Fanuc TP program (LS listing): CODE1_1.ls

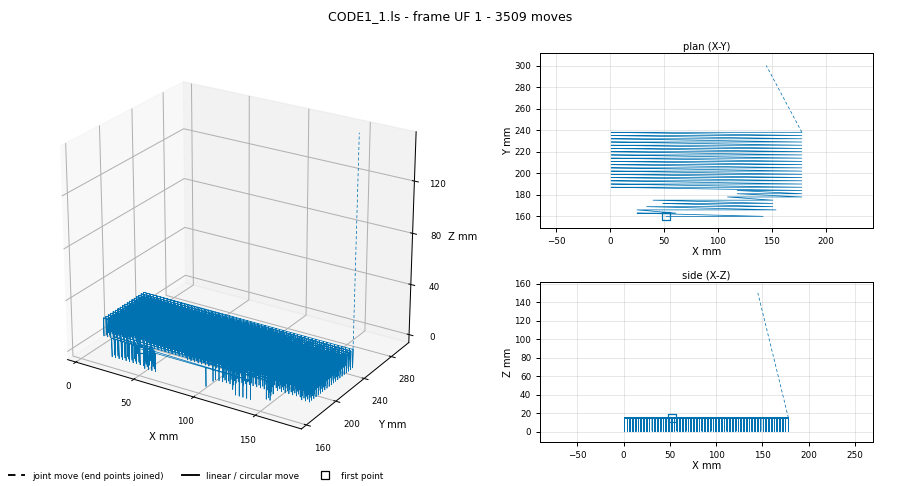
[picture p0: tool path of CODE1_1.ls in frame UF 1, 3509 of 3509 moves have a stored position in this frame; points joined in program order, loops and branches not executed]
/PROG CODE1_1
/ATTR
OWNER		= NOC_FANU;
COMMENT		= "NOC_FANUC";
PROG_SIZE	= 328;
CREATE		= DATE 97-07-08  TIME 03:05:20;
MODIFIED	= DATE 17-07-08  TIME 03:05:26;
FILE_NAME	= ;
VERSION		= 0;
LINE_COUNT	= 10;
MEMORY_SIZE	= 692;
PROTECT		= READ_WRITE;
TCD:  STACK_SIZE	= 0,
      TASK_PRIORITY	= 0,
      TIME_SLICE	= 0,
      BUSY_LAMP_OFF	= 0,
      ABORT_REQUEST	= 0,
      PAUSE_REQUEST	= 0;
DEFAULT_GROUP	= 1,*,*,*,*;
CONTROL_CODE	= 00000000 00000000;
/APPL
/MN
1:UFRAME_NUM=1 ;
2:UTOOL_NUM=1;
3:J P[7599] 10% CNT100;
4:L P[7600] 250mm/sec CNT100;
5:L P[7601] 250mm/sec FINE;
6:L P[7602] 250mm/sec CNT100;
7:L P[7603] 250mm/sec CNT100;
8:L P[7604] 250mm/sec FINE;
9:L P[7605] 250mm/sec CNT100;
10:L P[7606] 250mm/sec CNT100;
11:L P[7607] 250mm/sec FINE;
12:L P[7608] 250mm/sec CNT100;
13:L P[7609] 250mm/sec CNT100;
14:L P[7610] 250mm/sec FINE;
15:L P[7611] 250mm/sec CNT100;
16:L P[7612] 250mm/sec CNT100;
17:L P[7613] 250mm/sec FINE;
18:L P[7614] 250mm/sec CNT100;
19:L P[7636] 250mm/sec CNT100;
20:L P[7637] 250mm/sec FINE;
21:L P[7638] 250mm/sec CNT100;
22:L P[7639] 250mm/sec CNT100;
23:L P[7640] 250mm/sec FINE;
24:L P[7641] 250mm/sec CNT100;
25:L P[7642] 250mm/sec CNT100;
26:L P[7643] 250mm/sec FINE;
27:L P[7644] 250mm/sec CNT100;
28:L P[7645] 250mm/sec CNT100;
29:L P[7646] 250mm/sec FINE;
30:L P[7647] 250mm/sec CNT100;
31:L P[7648] 250mm/sec CNT100;
32:L P[7649] 250mm/sec FINE;
33:L P[7650] 250mm/sec CNT100;
34:L P[7666] 250mm/sec CNT100;
35:L P[7667] 250mm/sec FINE;
36:L P[7668] 250mm/sec CNT100;
37:L P[7669] 250mm/sec CNT100;
38:L P[7670] 250mm/sec FINE;
39:L P[7671] 250mm/sec CNT100;
40:L P[7672] 250mm/sec CNT100;
41:L P[7673] 250mm/sec FINE;
42:L P[7674] 250mm/sec CNT100;
43:L P[7675] 250mm/sec CNT100;
44:L P[7676] 250mm/sec FINE;
45:L P[7677] 250mm/sec CNT100;
46:L P[7678] 250mm/sec CNT100;
47:L P[7679] 250mm/sec FINE;
48:L P[7680] 250mm/sec CNT100;
49:L P[7681] 250mm/sec CNT100;
50:L P[7682] 250mm/sec FINE;
51:L P[7683] 250mm/sec CNT100;
52:L P[7684] 250mm/sec CNT100;
53:L P[7685] 250mm/sec FINE;
54:L P[7686] 250mm/sec CNT100;
55:L P[7687] 250mm/sec CNT100;
56:L P[7688] 250mm/sec FINE;
57:L P[7689] 250mm/sec CNT100;
58:L P[7690] 250mm/sec CNT100;
59:L P[7691] 250mm/sec FINE;
60:L P[7692] 250mm/sec CNT100;
61:L P[7693] 250mm/sec CNT100;
62:L P[7694] 250mm/sec FINE;
63:L P[7695] 250mm/sec CNT100;
64:L P[7696] 250mm/sec CNT100;
65:L P[7697] 250mm/sec FINE;
66:L P[7698] 250mm/sec CNT100;
67:L P[7702] 250mm/sec CNT100;
68:L P[7703] 250mm/sec FINE;
69:L P[7704] 250mm/sec CNT100;
70:L P[7756] 250mm/sec CNT100;
71:L P[7757] 250mm/sec FINE;
72:L P[7758] 250mm/sec CNT100;
73:L P[7759] 250mm/sec CNT100;
74:L P[7760] 250mm/sec FINE;
75:L P[7761] 250mm/sec CNT100;
76:L P[7762] 250mm/sec CNT100;
77:L P[7763] 250mm/sec FINE;
78:L P[7764] 250mm/sec CNT100;
79:L P[7765] 250mm/sec CNT100;
80:L P[7766] 250mm/sec FINE;
81:L P[7767] 250mm/sec CNT100;
82:L P[7768] 250mm/sec CNT100;
83:L P[7769] 250mm/sec FINE;
84:L P[7770] 250mm/sec CNT100;
85:L P[7771] 250mm/sec CNT100;
86:L P[7772] 250mm/sec FINE;
87:L P[7773] 250mm/sec CNT100;
88:L P[7774] 250mm/sec CNT100;
89:L P[7775] 250mm/sec FINE;
90:L P[7776] 250mm/sec CNT100;
91:L P[7777] 250mm/sec CNT100;
92:L P[7778] 250mm/sec FINE;
93:L P[7779] 250mm/sec CNT100;
94:L P[7783] 250mm/sec CNT100;
95:L P[7784] 250mm/sec FINE;
96:L P[7785] 250mm/sec CNT100;
97:L P[7786] 250mm/sec CNT100;
98:L P[7787] 250mm/sec FINE;
99:L P[7788] 250mm/sec CNT100;
100:L P[7789] 250mm/sec CNT100;
101:L P[7790] 250mm/sec FINE;
102:L P[7791] 250mm/sec CNT100;
103:L P[7810] 250mm/sec CNT100;
104:L P[7811] 250mm/sec FINE;
105:L P[7812] 250mm/sec CNT100;
106:L P[7837] 250mm/sec CNT100;
107:L P[7838] 250mm/sec FINE;
108:L P[7839] 250mm/sec CNT100;
109:L P[7840] 250mm/sec CNT100;
110:L P[7841] 250mm/sec FINE;
111:L P[7842] 250mm/sec CNT100;
112:L P[7849] 250mm/sec CNT100;
113:L P[7850] 250mm/sec FINE;
114:L P[7851] 250mm/sec CNT100;
115:L P[7855] 250mm/sec CNT100;
116:L P[7856] 250mm/sec FINE;
117:L P[7857] 250mm/sec CNT100;
118:L P[7864] 250mm/sec CNT100;
119:L P[7865] 250mm/sec FINE;
120:L P[7866] 250mm/sec CNT100;
121:L P[7870] 250mm/sec CNT100;
122:L P[7871] 250mm/sec FINE;
123:L P[7872] 250mm/sec CNT100;
124:L P[7873] 250mm/sec CNT100;
125:L P[7874] 250mm/sec FINE;
126:L P[7875] 250mm/sec CNT100;
127:L P[7918] 250mm/sec CNT100;
128:L P[7919] 250mm/sec FINE;
129:L P[7920] 250mm/sec CNT100;
130:L P[7939] 250mm/sec CNT100;
131:L P[7940] 250mm/sec FINE;
132:L P[7941] 250mm/sec CNT100;
133:L P[7942] 250mm/sec CNT100;
134:L P[7943] 250mm/sec FINE;
135:L P[7944] 250mm/sec CNT100;
136:L P[7945] 250mm/sec CNT100;
137:L P[7946] 250mm/sec FINE;
138:L P[7947] 250mm/sec CNT100;
139:L P[7948] 250mm/sec CNT100;
140:L P[7949] 250mm/sec FINE;
141:L P[7950] 250mm/sec CNT100;
142:L P[7951] 250mm/sec CNT100;
143:L P[7952] 250mm/sec FINE;
144:L P[7953] 250mm/sec CNT100;
145:L P[7954] 250mm/sec CNT100;
146:L P[7955] 250mm/sec FINE;
147:L P[7956] 250mm/sec CNT100;
148:L P[7957] 250mm/sec CNT100;
149:L P[7958] 250mm/sec FINE;
150:L P[7959] 250mm/sec CNT100;
151:L P[7960] 250mm/sec CNT100;
152:L P[7961] 250mm/sec FINE;
153:L P[7962] 250mm/sec CNT100;
154:L P[7990] 250mm/sec CNT100;
155:L P[7991] 250mm/sec FINE;
156:L P[7992] 250mm/sec CNT100;
157:L P[7999] 250mm/sec CNT100;
158:L P[8000] 250mm/sec FINE;
159:L P[8001] 250mm/sec CNT100;
160:L P[8014] 250mm/sec CNT100;
161:L P[8015] 250mm/sec FINE;
162:L P[8016] 250mm/sec CNT100;
163:L P[8017] 250mm/sec CNT100;
164:L P[8018] 250mm/sec FINE;
165:L P[8019] 250mm/sec CNT100;
166:L P[8020] 250mm/sec CNT100;
167:L P[8021] 250mm/sec FINE;
168:L P[8022] 250mm/sec CNT100;
169:L P[8023] 250mm/sec CNT100;
170:L P[8024] 250mm/sec FINE;
171:L P[8025] 250mm/sec CNT100;
172:L P[8026] 250mm/sec CNT100;
173:L P[8027] 250mm/sec FINE;
174:L P[8028] 250mm/sec CNT100;
175:L P[8029] 250mm/sec CNT100;
176:L P[8030] 250mm/sec FINE;
177:L P[8031] 250mm/sec CNT100;
178:L P[8050] 250mm/sec CNT100;
179:L P[8051] 250mm/sec FINE;
180:L P[8052] 250mm/sec CNT100;
181:L P[8053] 250mm/sec CNT100;
182:L P[8054] 250mm/sec FINE;
183:L P[8055] 250mm/sec CNT100;
184:L P[8074] 250mm/sec CNT100;
185:L P[8075] 250mm/sec FINE;
186:L P[8076] 250mm/sec CNT100;
187:L P[8080] 250mm/sec CNT100;
188:L P[8081] 250mm/sec FINE;
189:L P[8082] 250mm/sec CNT100;
190:L P[8083] 250mm/sec CNT100;
191:L P[8084] 250mm/sec FINE;
192:L P[8085] 250mm/sec CNT100;
193:L P[8086] 250mm/sec CNT100;
194:L P[8087] 250mm/sec FINE;
195:L P[8088] 250mm/sec CNT100;
196:L P[8089] 250mm/sec CNT100;
197:L P[8090] 250mm/sec FINE;
198:L P[8091] 250mm/sec CNT100;
199:L P[8092] 250mm/sec CNT100;
200:L P[8093] 250mm/sec FINE;
201:L P[8094] 250mm/sec CNT100;
202:L P[8095] 250mm/sec CNT100;
203:L P[8096] 250mm/sec FINE;
204:L P[8097] 250mm/sec CNT100;
205:L P[8098] 250mm/sec CNT100;
206:L P[8099] 250mm/sec FINE;
207:L P[8100] 250mm/sec CNT100;
208:L P[8101] 250mm/sec CNT100;
209:L P[8102] 250mm/sec FINE;
210:L P[8103] 250mm/sec CNT100;
211:L P[8104] 250mm/sec CNT100;
212:L P[8105] 250mm/sec FINE;
213:L P[8106] 250mm/sec CNT100;
214:L P[8107] 250mm/sec CNT100;
215:L P[8108] 250mm/sec FINE;
216:L P[8109] 250mm/sec CNT100;
217:L P[8110] 250mm/sec CNT100;
218:L P[8111] 250mm/sec FINE;
219:L P[8112] 250mm/sec CNT100;
220:L P[8113] 250mm/sec CNT100;
221:L P[8114] 250mm/sec FINE;
222:L P[8115] 250mm/sec CNT100;
223:L P[8125] 250mm/sec CNT100;
224:L P[8126] 250mm/sec FINE;
225:L P[8127] 250mm/sec CNT100;
226:L P[8128] 250mm/sec CNT100;
227:L P[8129] 250mm/sec FINE;
228:L P[8130] 250mm/sec CNT100;
229:L P[8131] 250mm/sec CNT100;
230:L P[8132] 250mm/sec FINE;
231:L P[8133] 250mm/sec CNT100;
232:L P[8167] 250mm/sec CNT100;
233:L P[8168] 250mm/sec FINE;
234:L P[8169] 250mm/sec CNT100;
235:L P[8173] 250mm/sec CNT100;
236:L P[8174] 250mm/sec FINE;
237:L P[8175] 250mm/sec CNT100;
238:L P[8176] 250mm/sec CNT100;
239:L P[8177] 250mm/sec FINE;
240:L P[8178] 250mm/sec CNT100;
241:L P[8179] 250mm/sec CNT100;
242:L P[8180] 250mm/sec FINE;
243:L P[8181] 250mm/sec CNT100;
244:L P[8182] 250mm/sec CNT100;
245:L P[8183] 250mm/sec FINE;
246:L P[8184] 250mm/sec CNT100;
247:L P[8185] 250mm/sec CNT100;
248:L P[8186] 250mm/sec FINE;
249:L P[8187] 250mm/sec CNT100;
250:L P[8188] 250mm/sec CNT100;
251:L P[8189] 250mm/sec FINE;
252:L P[8190] 250mm/sec CNT100;
253:L P[8194] 250mm/sec CNT100;
254:L P[8195] 250mm/sec FINE;
255:L P[8196] 250mm/sec CNT100;
256:L P[8200] 250mm/sec CNT100;
257:L P[8201] 250mm/sec FINE;
258:L P[8202] 250mm/sec CNT100;
259:L P[8203] 250mm/sec CNT100;
260:L P[8204] 250mm/sec FINE;
261:L P[8205] 250mm/sec CNT100;
262:L P[8206] 250mm/sec CNT100;
263:L P[8207] 250mm/sec FINE;
264:L P[8208] 250mm/sec CNT100;
265:L P[8209] 250mm/sec CNT100;
266:L P[8210] 250mm/sec FINE;
267:L P[8211] 250mm/sec CNT100;
268:L P[8212] 250mm/sec CNT100;
269:L P[8213] 250mm/sec FINE;
270:L P[8214] 250mm/sec CNT100;
271:L P[8215] 250mm/sec CNT100;
272:L P[8216] 250mm/sec FINE;
273:L P[8217] 250mm/sec CNT100;
274:L P[8218] 250mm/sec CNT100;
275:L P[8219] 250mm/sec FINE;
276:L P[8220] 250mm/sec CNT100;
277:L P[8221] 250mm/sec CNT100;
278:L P[8222] 250mm/sec FINE;
279:L P[8223] 250mm/sec CNT100;
280:L P[8224] 250mm/sec CNT100;
281:L P[8225] 250mm/sec FINE;
282:L P[8226] 250mm/sec CNT100;
283:L P[8227] 250mm/sec CNT100;
284:L P[8228] 250mm/sec FINE;
285:L P[8229] 250mm/sec CNT100;
286:L P[8269] 250mm/sec CNT100;
287:L P[8270] 250mm/sec FINE;
288:L P[8271] 250mm/sec CNT100;
289:L P[8272] 250mm/sec CNT100;
290:L P[8273] 250mm/sec FINE;
291:L P[8274] 250mm/sec CNT100;
292:L P[8278] 250mm/sec CNT100;
293:L P[8279] 250mm/sec FINE;
294:L P[8280] 250mm/sec CNT100;
295:L P[8290] 250mm/sec CNT100;
296:L P[8291] 250mm/sec FINE;
297:L P[8292] 250mm/sec CNT100;
298:L P[8296] 250mm/sec CNT100;
299:L P[8297] 250mm/sec FINE;
300:L P[8298] 250mm/sec CNT100;
301:L P[8299] 250mm/sec CNT100;
302:L P[8300] 250mm/sec FINE;
303:L P[8301] 250mm/sec CNT100;
304:L P[8302] 250mm/sec CNT100;
305:L P[8303] 250mm/sec FINE;
306:L P[8304] 250mm/sec CNT100;
307:L P[8305] 250mm/sec CNT100;
308:L P[8306] 250mm/sec FINE;
309:L P[8307] 250mm/sec CNT100;
310:L P[8308] 250mm/sec CNT100;
311:L P[8309] 250mm/sec FINE;
312:L P[8310] 250mm/sec CNT100;
313:L P[8311] 250mm/sec CNT100;
314:L P[8312] 250mm/sec FINE;
315:L P[8313] 250mm/sec CNT100;
316:L P[8314] 250mm/sec CNT100;
317:L P[8315] 250mm/sec FINE;
318:L P[8316] 250mm/sec CNT100;
319:L P[8317] 250mm/sec CNT100;
320:L P[8318] 250mm/sec FINE;
321:L P[8319] 250mm/sec CNT100;
322:L P[8320] 250mm/sec CNT100;
323:L P[8321] 250mm/sec FINE;
324:L P[8322] 250mm/sec CNT100;
325:L P[8323] 250mm/sec CNT100;
326:L P[8324] 250mm/sec FINE;
327:L P[8325] 250mm/sec CNT100;
328:L P[8326] 250mm/sec CNT100;
329:L P[8327] 250mm/sec FINE;
330:L P[8328] 250mm/sec CNT100;
331:L P[8329] 250mm/sec CNT100;
332:L P[8330] 250mm/sec FINE;
333:L P[8331] 250mm/sec CNT100;
334:L P[8332] 250mm/sec CNT100;
335:L P[8333] 250mm/sec FINE;
336:L P[8334] 250mm/sec CNT100;
337:L P[8335] 250mm/sec CNT100;
338:L P[8336] 250mm/sec FINE;
339:L P[8337] 250mm/sec CNT100;
340:L P[8338] 250mm/sec CNT100;
341:L P[8339] 250mm/sec FINE;
342:L P[8340] 250mm/sec CNT100;
343:L P[8341] 250mm/sec CNT100;
344:L P[8342] 250mm/sec FINE;
345:L P[8343] 250mm/sec CNT100;
346:L P[8344] 250mm/sec CNT100;
347:L P[8345] 250mm/sec FINE;
348:L P[8346] 250mm/sec CNT100;
349:L P[8347] 250mm/sec CNT100;
350:L P[8348] 250mm/sec FINE;
351:L P[8349] 250mm/sec CNT100;
352:L P[8350] 250mm/sec CNT100;
353:L P[8351] 250mm/sec FINE;
354:L P[8352] 250mm/sec CNT100;
355:L P[8353] 250mm/sec CNT100;
356:L P[8354] 250mm/sec FINE;
357:L P[8355] 250mm/sec CNT100;
358:L P[8401] 250mm/sec CNT100;
359:L P[8402] 250mm/sec FINE;
360:L P[8403] 250mm/sec CNT100;
361:L P[8404] 250mm/sec CNT100;
362:L P[8405] 250mm/sec FINE;
363:L P[8406] 250mm/sec CNT100;
364:L P[8407] 250mm/sec CNT100;
365:L P[8408] 250mm/sec FINE;
366:L P[8409] 250mm/sec CNT100;
367:L P[8410] 250mm/sec CNT100;
368:L P[8411] 250mm/sec FINE;
369:L P[8412] 250mm/sec CNT100;
370:L P[8413] 250mm/sec CNT100;
371:L P[8414] 250mm/sec FINE;
372:L P[8415] 250mm/sec CNT100;
373:L P[8416] 250mm/sec CNT100;
374:L P[8417] 250mm/sec FINE;
375:L P[8418] 250mm/sec CNT100;
376:L P[8419] 250mm/sec CNT100;
377:L P[8420] 250mm/sec FINE;
378:L P[8421] 250mm/sec CNT100;
379:L P[8422] 250mm/sec CNT100;
380:L P[8423] 250mm/sec FINE;
381:L P[8424] 250mm/sec CNT100;
382:L P[8425] 250mm/sec CNT100;
383:L P[8426] 250mm/sec FINE;
384:L P[8427] 250mm/sec CNT100;
385:L P[8428] 250mm/sec CNT100;
386:L P[8429] 250mm/sec FINE;
387:L P[8430] 250mm/sec CNT100;
388:L P[8431] 250mm/sec CNT100;
389:L P[8432] 250mm/sec FINE;
390:L P[8433] 250mm/sec CNT100;
391:L P[8434] 250mm/sec CNT100;
392:L P[8435] 250mm/sec FINE;
393:L P[8436] 250mm/sec CNT100;
394:L P[8437] 250mm/sec CNT100;
395:L P[8438] 250mm/sec FINE;
396:L P[8439] 250mm/sec CNT100;
397:L P[8440] 250mm/sec CNT100;
398:L P[8441] 250mm/sec FINE;
399:L P[8442] 250mm/sec CNT100;
400:L P[8443] 250mm/sec CNT100;
401:L P[8444] 250mm/sec FINE;
402:L P[8445] 250mm/sec CNT100;
403:L P[8446] 250mm/sec CNT100;
404:L P[8447] 250mm/sec FINE;
405:L P[8448] 250mm/sec CNT100;
406:L P[8458] 250mm/sec CNT100;
407:L P[8459] 250mm/sec FINE;
408:L P[8460] 250mm/sec CNT100;
409:L P[8467] 250mm/sec CNT100;
410:L P[8468] 250mm/sec FINE;
411:L P[8469] 250mm/sec CNT100;
412:L P[8470] 250mm/sec CNT100;
413:L P[8471] 250mm/sec FINE;
414:L P[8472] 250mm/sec CNT100;
415:L P[8473] 250mm/sec CNT100;
416:L P[8474] 250mm/sec FINE;
417:L P[8475] 250mm/sec CNT100;
418:L P[8476] 250mm/sec CNT100;
419:L P[8477] 250mm/sec FINE;
420:L P[8478] 250mm/sec CNT100;
421:L P[8479] 250mm/sec CNT100;
422:L P[8480] 250mm/sec FINE;
423:L P[8481] 250mm/sec CNT100;
424:L P[8482] 250mm/sec CNT100;
425:L P[8483] 250mm/sec FINE;
426:L P[8484] 250mm/sec CNT100;
427:L P[8485] 250mm/sec CNT100;
428:L P[8486] 250mm/sec FINE;
429:L P[8487] 250mm/sec CNT100;
430:L P[8488] 250mm/sec CNT100;
431:L P[8489] 250mm/sec FINE;
432:L P[8490] 250mm/sec CNT100;
433:L P[8491] 250mm/sec CNT100;
434:L P[8492] 250mm/sec FINE;
435:L P[8493] 250mm/sec CNT100;
436:L P[8494] 250mm/sec CNT100;
437:L P[8495] 250mm/sec FINE;
438:L P[8496] 250mm/sec CNT100;
439:L P[8497] 250mm/sec CNT100;
440:L P[8498] 250mm/sec FINE;
441:L P[8499] 250mm/sec CNT100;
442:L P[8500] 250mm/sec CNT100;
443:L P[8501] 250mm/sec FINE;
444:L P[8502] 250mm/sec CNT100;
445:L P[8503] 250mm/sec CNT100;
446:L P[8504] 250mm/sec FINE;
447:L P[8505] 250mm/sec CNT100;
448:L P[8506] 250mm/sec CNT100;
449:L P[8507] 250mm/sec FINE;
450:L P[8508] 250mm/sec CNT100;
451:L P[8509] 250mm/sec CNT100;
452:L P[8510] 250mm/sec FINE;
453:L P[8511] 250mm/sec CNT100;
454:L P[8512] 250mm/sec CNT100;
455:L P[8513] 250mm/sec FINE;
456:L P[8514] 250mm/sec CNT100;
457:L P[8515] 250mm/sec CNT100;
458:L P[8516] 250mm/sec FINE;
459:L P[8517] 250mm/sec CNT100;
460:L P[8518] 250mm/sec CNT100;
461:L P[8519] 250mm/sec FINE;
462:L P[8520] 250mm/sec CNT100;
463:L P[8521] 250mm/sec CNT100;
464:L P[8522] 250mm/sec FINE;
465:L P[8523] 250mm/sec CNT100;
466:L P[8524] 250mm/sec CNT100;
467:L P[8525] 250mm/sec FINE;
468:L P[8526] 250mm/sec CNT100;
469:L P[8527] 250mm/sec CNT100;
470:L P[8528] 250mm/sec FINE;
471:L P[8529] 250mm/sec CNT100;
472:L P[8530] 250mm/sec CNT100;
473:L P[8531] 250mm/sec FINE;
474:L P[8532] 250mm/sec CNT100;
475:L P[8533] 250mm/sec CNT100;
476:L P[8534] 250mm/sec FINE;
477:L P[8535] 250mm/sec CNT100;
478:L P[8536] 250mm/sec CNT100;
479:L P[8537] 250mm/sec FINE;
480:L P[8538] 250mm/sec CNT100;
481:L P[8539] 250mm/sec CNT100;
482:L P[8540] 250mm/sec FINE;
483:L P[8541] 250mm/sec CNT100;
484:L P[8542] 250mm/sec CNT100;
485:L P[8543] 250mm/sec FINE;
486:L P[8544] 250mm/sec CNT100;
487:L P[8545] 250mm/sec CNT100;
488:L P[8546] 250mm/sec FINE;
489:L P[8547] 250mm/sec CNT100;
490:L P[8548] 250mm/sec CNT100;
491:L P[8549] 250mm/sec FINE;
492:L P[8550] 250mm/sec CNT100;
493:L P[8551] 250mm/sec CNT100;
494:L P[8552] 250mm/sec FINE;
495:L P[8553] 250mm/sec CNT100;
496:L P[8554] 250mm/sec CNT100;
497:L P[8555] 250mm/sec FINE;
498:L P[8556] 250mm/sec CNT100;
499:L P[8557] 250mm/sec CNT100;
500:L P[8558] 250mm/sec FINE;
501:L P[8559] 250mm/sec CNT100;
502:L P[8560] 250mm/sec CNT100;
503:L P[8561] 250mm/sec FINE;
504:L P[8562] 250mm/sec CNT100;
505:L P[8563] 250mm/sec CNT100;
506:L P[8564] 250mm/sec FINE;
507:L P[8565] 250mm/sec CNT100;
508:L P[8566] 250mm/sec CNT100;
509:L P[8567] 250mm/sec FINE;
510:L P[8568] 250mm/sec CNT100;
511:L P[8569] 250mm/sec CNT100;
512:L P[8570] 250mm/sec FINE;
513:L P[8571] 250mm/sec CNT100;
514:L P[8572] 250mm/sec CNT100;
515:L P[8573] 250mm/sec FINE;
516:L P[8574] 250mm/sec CNT100;
517:L P[8575] 250mm/sec CNT100;
518:L P[8576] 250mm/sec FINE;
519:L P[8577] 250mm/sec CNT100;
520:L P[8578] 250mm/sec CNT100;
521:L P[8579] 250mm/sec FINE;
522:L P[8580] 250mm/sec CNT100;
523:L P[8581] 250mm/sec CNT100;
524:L P[8582] 250mm/sec FINE;
525:L P[8583] 250mm/sec CNT100;
526:L P[8584] 250mm/sec CNT100;
527:L P[8585] 250mm/sec FINE;
528:L P[8586] 250mm/sec CNT100;
529:L P[8587] 250mm/sec CNT100;
530:L P[8588] 250mm/sec FINE;
531:L P[8589] 250mm/sec CNT100;
532:L P[8590] 250mm/sec CNT100;
533:L P[8591] 250mm/sec FINE;
534:L P[8592] 250mm/sec CNT100;
535:L P[8593] 250mm/sec CNT100;
536:L P[8594] 250mm/sec FINE;
537:L P[8595] 250mm/sec CNT100;
538:L P[8596] 250mm/sec CNT100;
539:L P[8597] 250mm/sec FINE;
540:L P[8598] 250mm/sec CNT100;
541:L P[8599] 250mm/sec CNT100;
542:L P[8600] 250mm/sec FINE;
543:L P[8601] 250mm/sec CNT100;
544:L P[8602] 250mm/sec CNT100;
545:L P[8603] 250mm/sec FINE;
546:L P[8604] 250mm/sec CNT100;
547:L P[8605] 250mm/sec CNT100;
548:L P[8606] 250mm/sec FINE;
549:L P[8607] 250mm/sec CNT100;
550:L P[8608] 250mm/sec CNT100;
551:L P[8609] 250mm/sec FINE;
552:L P[8610] 250mm/sec CNT100;
553:L P[8611] 250mm/sec CNT100;
554:L P[8612] 250mm/sec FINE;
555:L P[8613] 250mm/sec CNT100;
556:L P[8614] 250mm/sec CNT100;
557:L P[8615] 250mm/sec FINE;
558:L P[8616] 250mm/sec CNT100;
559:L P[8617] 250mm/sec CNT100;
560:L P[8618] 250mm/sec FINE;
561:L P[8619] 250mm/sec CNT100;
562:L P[8620] 250mm/sec CNT100;
563:L P[8621] 250mm/sec FINE;
564:L P[8622] 250mm/sec CNT100;
565:L P[8623] 250mm/sec CNT100;
566:L P[8624] 250mm/sec FINE;
567:L P[8625] 250mm/sec CNT100;
568:L P[8626] 250mm/sec CNT100;
569:L P[8627] 250mm/sec FINE;
570:L P[8628] 250mm/sec CNT100;
571:L P[8629] 250mm/sec CNT100;
572:L P[8630] 250mm/sec FINE;
573:L P[8631] 250mm/sec CNT100;
574:L P[8632] 250mm/sec CNT100;
575:L P[8633] 250mm/sec FINE;
576:L P[8634] 250mm/sec CNT100;
577:L P[8635] 250mm/sec CNT100;
578:L P[8636] 250mm/sec FINE;
579:L P[8637] 250mm/sec CNT100;
580:L P[8638] 250mm/sec CNT100;
581:L P[8639] 250mm/sec FINE;
582:L P[8640] 250mm/sec CNT100;
583:L P[8641] 250mm/sec CNT100;
584:L P[8642] 250mm/sec FINE;
585:L P[8643] 250mm/sec CNT100;
586:L P[8644] 250mm/sec CNT100;
587:L P[8645] 250mm/sec FINE;
588:L P[8646] 250mm/sec CNT100;
589:L P[8647] 250mm/sec CNT100;
590:L P[8648] 250mm/sec FINE;
591:L P[8649] 250mm/sec CNT100;
592:L P[8650] 250mm/sec CNT100;
593:L P[8651] 250mm/sec FINE;
594:L P[8652] 250mm/sec CNT100;
595:L P[8653] 250mm/sec CNT100;
596:L P[8654] 250mm/sec FINE;
597:L P[8655] 250mm/sec CNT100;
598:L P[8656] 250mm/sec CNT100;
599:L P[8657] 250mm/sec FINE;
600:L P[8658] 250mm/sec CNT100;
601:L P[8659] 250mm/sec CNT100;
602:L P[8660] 250mm/sec FINE;
603:L P[8661] 250mm/sec CNT100;
604:L P[8662] 250mm/sec CNT100;
605:L P[8663] 250mm/sec FINE;
606:L P[8664] 250mm/sec CNT100;
607:L P[8665] 250mm/sec CNT100;
608:L P[8666] 250mm/sec FINE;
609:L P[8667] 250mm/sec CNT100;
610:L P[8668] 250mm/sec CNT100;
611:L P[8669] 250mm/sec FINE;
612:L P[8670] 250mm/sec CNT100;
613:L P[8671] 250mm/sec CNT100;
614:L P[8672] 250mm/sec FINE;
615:L P[8673] 250mm/sec CNT100;
616:L P[8674] 250mm/sec CNT100;
617:L P[8675] 250mm/sec FINE;
618:L P[8676] 250mm/sec CNT100;
619:L P[8677] 250mm/sec CNT100;
620:L P[8678] 250mm/sec FINE;
621:L P[8679] 250mm/sec CNT100;
622:L P[8680] 250mm/sec CNT100;
623:L P[8681] 250mm/sec FINE;
624:L P[8682] 250mm/sec CNT100;
625:L P[8683] 250mm/sec CNT100;
626:L P[8684] 250mm/sec FINE;
627:L P[8685] 250mm/sec CNT100;
628:L P[8686] 250mm/sec CNT100;
629:L P[8687] 250mm/sec FINE;
630:L P[8688] 250mm/sec CNT100;
631:L P[8689] 250mm/sec CNT100;
632:L P[8690] 250mm/sec FINE;
633:L P[8691] 250mm/sec CNT100;
634:L P[8692] 250mm/sec CNT100;
635:L P[8693] 250mm/sec FINE;
636:L P[8694] 250mm/sec CNT100;
637:L P[8695] 250mm/sec CNT100;
638:L P[8696] 250mm/sec FINE;
639:L P[8697] 250mm/sec CNT100;
640:L P[8698] 250mm/sec CNT100;
641:L P[8699] 250mm/sec FINE;
642:L P[8700] 250mm/sec CNT100;
643:L P[8701] 250mm/sec CNT100;
644:L P[8702] 250mm/sec FINE;
645:L P[8703] 250mm/sec CNT100;
646:L P[8704] 250mm/sec CNT100;
647:L P[8705] 250mm/sec FINE;
648:L P[8706] 250mm/sec CNT100;
649:L P[8707] 250mm/sec CNT100;
650:L P[8708] 250mm/sec FINE;
651:L P[8709] 250mm/sec CNT100;
652:L P[8710] 250mm/sec CNT100;
653:L P[8711] 250mm/sec FINE;
654:L P[8712] 250mm/sec CNT100;
655:L P[8713] 250mm/sec CNT100;
656:L P[8714] 250mm/sec FINE;
657:L P[8715] 250mm/sec CNT100;
658:L P[8716] 250mm/sec CNT100;
659:L P[8717] 250mm/sec FINE;
660:L P[8718] 250mm/sec CNT100;
661:L P[8719] 250mm/sec CNT100;
662:L P[8720] 250mm/sec FINE;
663:L P[8721] 250mm/sec CNT100;
664:L P[8722] 250mm/sec CNT100;
665:L P[8723] 250mm/sec FINE;
666:L P[8724] 250mm/sec CNT100;
667:L P[8725] 250mm/sec CNT100;
668:L P[8726] 250mm/sec FINE;
669:L P[8727] 250mm/sec CNT100;
670:L P[8728] 250mm/sec CNT100;
671:L P[8729] 250mm/sec FINE;
672:L P[8730] 250mm/sec CNT100;
673:L P[8731] 250mm/sec CNT100;
674:L P[8732] 250mm/sec FINE;
675:L P[8733] 250mm/sec CNT100;
676:L P[8734] 250mm/sec CNT100;
677:L P[8735] 250mm/sec FINE;
678:L P[8736] 250mm/sec CNT100;
679:L P[8737] 250mm/sec CNT100;
680:L P[8738] 250mm/sec FINE;
681:L P[8739] 250mm/sec CNT100;
682:L P[8740] 250mm/sec CNT100;
683:L P[8741] 250mm/sec FINE;
684:L P[8742] 250mm/sec CNT100;
685:L P[8743] 250mm/sec CNT100;
686:L P[8744] 250mm/sec FINE;
687:L P[8745] 250mm/sec CNT100;
688:L P[8746] 250mm/sec CNT100;
689:L P[8747] 250mm/sec FINE;
690:L P[8748] 250mm/sec CNT100;
691:L P[8749] 250mm/sec CNT100;
692:L P[8750] 250mm/sec FINE;
693:L P[8751] 250mm/sec CNT100;
694:L P[8752] 250mm/sec CNT100;
695:L P[8753] 250mm/sec FINE;
696:L P[8754] 250mm/sec CNT100;
697:L P[8755] 250mm/sec CNT100;
698:L P[8756] 250mm/sec FINE;
699:L P[8757] 250mm/sec CNT100;
700:L P[8758] 250mm/sec CNT100;
701:L P[8759] 250mm/sec FINE;
702:L P[8760] 250mm/sec CNT100;
703:L P[8761] 250mm/sec CNT100;
704:L P[8762] 250mm/sec FINE;
705:L P[8763] 250mm/sec CNT100;
706:L P[8764] 250mm/sec CNT100;
707:L P[8765] 250mm/sec FINE;
708:L P[8766] 250mm/sec CNT100;
709:L P[8767] 250mm/sec CNT100;
710:L P[8768] 250mm/sec FINE;
711:L P[8769] 250mm/sec CNT100;
712:L P[8770] 250mm/sec CNT100;
713:L P[8771] 250mm/sec FINE;
714:L P[8772] 250mm/sec CNT100;
715:L P[8773] 250mm/sec CNT100;
716:L P[8774] 250mm/sec FINE;
717:L P[8775] 250mm/sec CNT100;
718:L P[8776] 250mm/sec CNT100;
719:L P[8777] 250mm/sec FINE;
720:L P[8778] 250mm/sec CNT100;
721:L P[8779] 250mm/sec CNT100;
722:L P[8780] 250mm/sec FINE;
723:L P[8781] 250mm/sec CNT100;
724:L P[8782] 250mm/sec CNT100;
725:L P[8783] 250mm/sec FINE;
726:L P[8784] 250mm/sec CNT100;
727:L P[8785] 250mm/sec CNT100;
728:L P[8786] 250mm/sec FINE;
729:L P[8787] 250mm/sec CNT100;
730:L P[8788] 250mm/sec CNT100;
731:L P[8789] 250mm/sec FINE;
732:L P[8790] 250mm/sec CNT100;
733:L P[8791] 250mm/sec CNT100;
734:L P[8792] 250mm/sec FINE;
735:L P[8793] 250mm/sec CNT100;
736:L P[8794] 250mm/sec CNT100;
737:L P[8795] 250mm/sec FINE;
738:L P[8796] 250mm/sec CNT100;
739:L P[8797] 250mm/sec CNT100;
740:L P[8798] 250mm/sec FINE;
741:L P[8799] 250mm/sec CNT100;
742:L P[8800] 250mm/sec CNT100;
743:L P[8801] 250mm/sec FINE;
744:L P[8802] 250mm/sec CNT100;
745:L P[8803] 250mm/sec CNT100;
746:L P[8804] 250mm/sec FINE;
747:L P[8805] 250mm/sec CNT100;
748:L P[8806] 250mm/sec CNT100;
749:L P[8807] 250mm/sec FINE;
750:L P[8808] 250mm/sec CNT100;
751:L P[8809] 250mm/sec CNT100;
752:L P[8810] 250mm/sec FINE;
753:L P[8811] 250mm/sec CNT100;
754:L P[8812] 250mm/sec CNT100;
755:L P[8813] 250mm/sec FINE;
756:L P[8814] 250mm/sec CNT100;
757:L P[8815] 250mm/sec CNT100;
758:L P[8816] 250mm/sec FINE;
759:L P[8817] 250mm/sec CNT100;
760:L P[8818] 250mm/sec CNT100;
761:L P[8819] 250mm/sec FINE;
762:L P[8820] 250mm/sec CNT100;
763:L P[8821] 250mm/sec CNT100;
764:L P[8822] 250mm/sec FINE;
765:L P[8823] 250mm/sec CNT100;
766:L P[8824] 250mm/sec CNT100;
767:L P[8825] 250mm/sec FINE;
768:L P[8826] 250mm/sec CNT100;
769:L P[8827] 250mm/sec CNT100;
770:L P[8828] 250mm/sec FINE;
771:L P[8829] 250mm/sec CNT100;
772:L P[8830] 250mm/sec CNT100;
773:L P[8831] 250mm/sec FINE;
774:L P[8832] 250mm/sec CNT100;
775:L P[8833] 250mm/sec CNT100;
776:L P[8834] 250mm/sec FINE;
777:L P[8835] 250mm/sec CNT100;
778:L P[8836] 250mm/sec CNT100;
779:L P[8837] 250mm/sec FINE;
780:L P[8838] 250mm/sec CNT100;
781:L P[8839] 250mm/sec CNT100;
782:L P[8840] 250mm/sec FINE;
783:L P[8841] 250mm/sec CNT100;
784:L P[8842] 250mm/sec CNT100;
785:L P[8843] 250mm/sec FINE;
786:L P[8844] 250mm/sec CNT100;
787:L P[8845] 250mm/sec CNT100;
788:L P[8846] 250mm/sec FINE;
789:L P[8847] 250mm/sec CNT100;
790:L P[8848] 250mm/sec CNT100;
791:L P[8849] 250mm/sec FINE;
792:L P[8850] 250mm/sec CNT100;
793:L P[8851] 250mm/sec CNT100;
794:L P[8852] 250mm/sec FINE;
795:L P[8853] 250mm/sec CNT100;
796:L P[8854] 250mm/sec CNT100;
797:L P[8855] 250mm/sec FINE;
798:L P[8856] 250mm/sec CNT100;
799:L P[8857] 250mm/sec CNT100;
800:L P[8858] 250mm/sec FINE;
801:L P[8859] 250mm/sec CNT100;
802:L P[8860] 250mm/sec CNT100;
803:L P[8861] 250mm/sec FINE;
804:L P[8862] 250mm/sec CNT100;
805:L P[8863] 250mm/sec CNT100;
806:L P[8864] 250mm/sec FINE;
807:L P[8865] 250mm/sec CNT100;
808:L P[8866] 250mm/sec CNT100;
809:L P[8867] 250mm/sec FINE;
810:L P[8868] 250mm/sec CNT100;
811:L P[8869] 250mm/sec CNT100;
812:L P[8870] 250mm/sec FINE;
813:L P[8871] 250mm/sec CNT100;
814:L P[8872] 250mm/sec CNT100;
815:L P[8873] 250mm/sec FINE;
816:L P[8874] 250mm/sec CNT100;
817:L P[8875] 250mm/sec CNT100;
818:L P[8876] 250mm/sec FINE;
819:L P[8877] 250mm/sec CNT100;
820:L P[8878] 250mm/sec CNT100;
821:L P[8879] 250mm/sec FINE;
822:L P[8880] 250mm/sec CNT100;
823:L P[8881] 250mm/sec CNT100;
824:L P[8882] 250mm/sec FINE;
825:L P[8883] 250mm/sec CNT100;
826:L P[8884] 250mm/sec CNT100;
827:L P[8885] 250mm/sec FINE;
828:L P[8886] 250mm/sec CNT100;
829:L P[8887] 250mm/sec CNT100;
830:L P[8888] 250mm/sec FINE;
831:L P[8889] 250mm/sec CNT100;
832:L P[8890] 250mm/sec CNT100;
833:L P[8891] 250mm/sec FINE;
834:L P[8892] 250mm/sec CNT100;
835:L P[8893] 250mm/sec CNT100;
836:L P[8894] 250mm/sec FINE;
837:L P[8895] 250mm/sec CNT100;
838:L P[8896] 250mm/sec CNT100;
839:L P[8897] 250mm/sec FINE;
840:L P[8898] 250mm/sec CNT100;
841:L P[8899] 250mm/sec CNT100;
842:L P[8900] 250mm/sec FINE;
843:L P[8901] 250mm/sec CNT100;
844:L P[8902] 250mm/sec CNT100;
845:L P[8903] 250mm/sec FINE;
846:L P[8904] 250mm/sec CNT100;
847:L P[8905] 250mm/sec CNT100;
848:L P[8906] 250mm/sec FINE;
849:L P[8907] 250mm/sec CNT100;
850:L P[8908] 250mm/sec CNT100;
851:L P[8909] 250mm/sec FINE;
852:L P[8910] 250mm/sec CNT100;
853:L P[8911] 250mm/sec CNT100;
854:L P[8912] 250mm/sec FINE;
855:L P[8913] 250mm/sec CNT100;
856:L P[8914] 250mm/sec CNT100;
857:L P[8915] 250mm/sec FINE;
858:L P[8916] 250mm/sec CNT100;
859:L P[8917] 250mm/sec CNT100;
860:L P[8918] 250mm/sec FINE;
861:L P[8919] 250mm/sec CNT100;
862:L P[8920] 250mm/sec CNT100;
863:L P[8921] 250mm/sec FINE;
864:L P[8922] 250mm/sec CNT100;
865:L P[8923] 250mm/sec CNT100;
866:L P[8924] 250mm/sec FINE;
867:L P[8925] 250mm/sec CNT100;
868:L P[8926] 250mm/sec CNT100;
869:L P[8927] 250mm/sec FINE;
870:L P[8928] 250mm/sec CNT100;
871:L P[8929] 250mm/sec CNT100;
872:L P[8930] 250mm/sec FINE;
873:L P[8931] 250mm/sec CNT100;
874:L P[8932] 250mm/sec CNT100;
875:L P[8933] 250mm/sec FINE;
876:L P[8934] 250mm/sec CNT100;
877:L P[8935] 250mm/sec CNT100;
878:L P[8936] 250mm/sec FINE;
879:L P[8937] 250mm/sec CNT100;
880:L P[8938] 250mm/sec CNT100;
881:L P[8939] 250mm/sec FINE;
882:L P[8940] 250mm/sec CNT100;
883:L P[8941] 250mm/sec CNT100;
884:L P[8942] 250mm/sec FINE;
885:L P[8943] 250mm/sec CNT100;
886:L P[8944] 250mm/sec CNT100;
887:L P[8945] 250mm/sec FINE;
888:L P[8946] 250mm/sec CNT100;
889:L P[8947] 250mm/sec CNT100;
890:L P[8948] 250mm/sec FINE;
891:L P[8949] 250mm/sec CNT100;
892:L P[8950] 250mm/sec CNT100;
893:L P[8951] 250mm/sec FINE;
894:L P[8952] 250mm/sec CNT100;
895:L P[8953] 250mm/sec CNT100;
896:L P[8954] 250mm/sec FINE;
897:L P[8955] 250mm/sec CNT100;
898:L P[8956] 250mm/sec CNT100;
899:L P[8957] 250mm/sec FINE;
900:L P[8958] 250mm/sec CNT100;
901:L P[8959] 250mm/sec CNT100;
902:L P[8960] 250mm/sec FINE;
903:L P[8961] 250mm/sec CNT100;
904:L P[8962] 250mm/sec CNT100;
905:L P[8963] 250mm/sec FINE;
906:L P[8964] 250mm/sec CNT100;
907:L P[8965] 250mm/sec CNT100;
908:L P[8966] 250mm/sec FINE;
909:L P[8967] 250mm/sec CNT100;
910:L P[8968] 250mm/sec CNT100;
911:L P[8969] 250mm/sec FINE;
912:L P[8970] 250mm/sec CNT100;
913:L P[8971] 250mm/sec CNT100;
914:L P[8972] 250mm/sec FINE;
915:L P[8973] 250mm/sec CNT100;
916:L P[8974] 250mm/sec CNT100;
917:L P[8975] 250mm/sec FINE;
918:L P[8976] 250mm/sec CNT100;
919:L P[8977] 250mm/sec CNT100;
920:L P[8978] 250mm/sec FINE;
921:L P[8979] 250mm/sec CNT100;
922:L P[8980] 250mm/sec CNT100;
923:L P[8981] 250mm/sec FINE;
924:L P[8982] 250mm/sec CNT100;
925:L P[8983] 250mm/sec CNT100;
926:L P[8984] 250mm/sec FINE;
927:L P[8985] 250mm/sec CNT100;
928:L P[8986] 250mm/sec CNT100;
929:L P[8987] 250mm/sec FINE;
930:L P[8988] 250mm/sec CNT100;
931:L P[8989] 250mm/sec CNT100;
932:L P[8990] 250mm/sec FINE;
933:L P[8991] 250mm/sec CNT100;
934:L P[8992] 250mm/sec CNT100;
935:L P[8993] 250mm/sec FINE;
936:L P[8994] 250mm/sec CNT100;
937:L P[8995] 250mm/sec CNT100;
938:L P[8996] 250mm/sec FINE;
939:L P[8997] 250mm/sec CNT100;
940:L P[8998] 250mm/sec CNT100;
941:L P[8999] 250mm/sec FINE;
942:L P[9000] 250mm/sec CNT100;
943:L P[9001] 250mm/sec CNT100;
944:L P[9002] 250mm/sec FINE;
945:L P[9003] 250mm/sec CNT100;
946:L P[9004] 250mm/sec CNT100;
947:L P[9005] 250mm/sec FINE;
948:L P[9006] 250mm/sec CNT100;
949:L P[9007] 250mm/sec CNT100;
950:L P[9008] 250mm/sec FINE;
951:L P[9009] 250mm/sec CNT100;
952:L P[9010] 250mm/sec CNT100;
953:L P[9011] 250mm/sec FINE;
954:L P[9012] 250mm/sec CNT100;
955:L P[9013] 250mm/sec CNT100;
956:L P[9014] 250mm/sec FINE;
957:L P[9015] 250mm/sec CNT100;
958:L P[9016] 250mm/sec CNT100;
959:L P[9017] 250mm/sec FINE;
960:L P[9018] 250mm/sec CNT100;
961:L P[9019] 250mm/sec CNT100;
962:L P[9020] 250mm/sec FINE;
963:L P[9021] 250mm/sec CNT100;
964:L P[9022] 250mm/sec CNT100;
965:L P[9023] 250mm/sec FINE;
966:L P[9024] 250mm/sec CNT100;
967:L P[9025] 250mm/sec CNT100;
968:L P[9026] 250mm/sec FINE;
969:L P[9027] 250mm/sec CNT100;
970:L P[9028] 250mm/sec CNT100;
971:L P[9029] 250mm/sec FINE;
972:L P[9030] 250mm/sec CNT100;
973:L P[9031] 250mm/sec CNT100;
974:L P[9032] 250mm/sec FINE;
975:L P[9033] 250mm/sec CNT100;
976:L P[9034] 250mm/sec CNT100;
977:L P[9035] 250mm/sec FINE;
978:L P[9036] 250mm/sec CNT100;
979:L P[9037] 250mm/sec CNT100;
980:L P[9038] 250mm/sec FINE;
981:L P[9039] 250mm/sec CNT100;
982:L P[9040] 250mm/sec CNT100;
983:L P[9041] 250mm/sec FINE;
984:L P[9042] 250mm/sec CNT100;
985:L P[9043] 250mm/sec CNT100;
986:L P[9044] 250mm/sec FINE;
987:L P[9045] 250mm/sec CNT100;
988:L P[9046] 250mm/sec CNT100;
989:L P[9047] 250mm/sec FINE;
990:L P[9048] 250mm/sec CNT100;
991:L P[9049] 250mm/sec CNT100;
992:L P[9050] 250mm/sec FINE;
993:L P[9051] 250mm/sec CNT100;
994:L P[9052] 250mm/sec CNT100;
995:L P[9053] 250mm/sec FINE;
996:L P[9054] 250mm/sec CNT100;
997:L P[9055] 250mm/sec CNT100;
998:L P[9056] 250mm/sec FINE;
999:L P[9057] 250mm/sec CNT100;
1000:L P[9058] 250mm/sec CNT100;
1001:L P[9059] 250mm/sec FINE;
1002:L P[9060] 250mm/sec CNT100;
1003:L P[9061] 250mm/sec CNT100;
1004:L P[9062] 250mm/sec FINE;
1005:L P[9063] 250mm/sec CNT100;
1006:L P[9064] 250mm/sec CNT100;
1007:L P[9065] 250mm/sec FINE;
1008:L P[9066] 250mm/sec CNT100;
1009:L P[9067] 250mm/sec CNT100;
1010:L P[9068] 250mm/sec FINE;
1011:L P[9069] 250mm/sec CNT100;
1012:L P[9070] 250mm/sec CNT100;
1013:L P[9071] 250mm/sec FINE;
1014:L P[9072] 250mm/sec CNT100;
1015:L P[9073] 250mm/sec CNT100;
1016:L P[9074] 250mm/sec FINE;
1017:L P[9075] 250mm/sec CNT100;
1018:L P[9076] 250mm/sec CNT100;
1019:L P[9077] 250mm/sec FINE;
1020:L P[9078] 250mm/sec CNT100;
1021:L P[9079] 250mm/sec CNT100;
1022:L P[9080] 250mm/sec FINE;
1023:L P[9081] 250mm/sec CNT100;
1024:L P[9082] 250mm/sec CNT100;
1025:L P[9083] 250mm/sec FINE;
1026:L P[9084] 250mm/sec CNT100;
1027:L P[9085] 250mm/sec CNT100;
1028:L P[9086] 250mm/sec FINE;
1029:L P[9087] 250mm/sec CNT100;
1030:L P[9088] 250mm/sec CNT100;
1031:L P[9089] 250mm/sec FINE;
1032:L P[9090] 250mm/sec CNT100;
1033:L P[9091] 250mm/sec CNT100;
1034:L P[9092] 250mm/sec FINE;
1035:L P[9093] 250mm/sec CNT100;
1036:L P[9094] 250mm/sec CNT100;
1037:L P[9095] 250mm/sec FINE;
1038:L P[9096] 250mm/sec CNT100;
1039:L P[9097] 250mm/sec CNT100;
1040:L P[9098] 250mm/sec FINE;
1041:L P[9099] 250mm/sec CNT100;
1042:L P[9100] 250mm/sec CNT100;
1043:L P[9101] 250mm/sec FINE;
1044:L P[9102] 250mm/sec CNT100;
1045:L P[9103] 250mm/sec CNT100;
1046:L P[9104] 250mm/sec FINE;
1047:L P[9105] 250mm/sec CNT100;
1048:L P[9106] 250mm/sec CNT100;
1049:L P[9107] 250mm/sec FINE;
1050:L P[9108] 250mm/sec CNT100;
1051:L P[9109] 250mm/sec CNT100;
1052:L P[9110] 250mm/sec FINE;
1053:L P[9111] 250mm/sec CNT100;
1054:L P[9112] 250mm/sec CNT100;
1055:L P[9113] 250mm/sec FINE;
1056:L P[9114] 250mm/sec CNT100;
1057:L P[9115] 250mm/sec CNT100;
1058:L P[9116] 250mm/sec FINE;
1059:L P[9117] 250mm/sec CNT100;
1060:L P[9118] 250mm/sec CNT100;
1061:L P[9119] 250mm/sec FINE;
1062:L P[9120] 250mm/sec CNT100;
1063:L P[9121] 250mm/sec CNT100;
1064:L P[9122] 250mm/sec FINE;
1065:L P[9123] 250mm/sec CNT100;
1066:L P[9124] 250mm/sec CNT100;
1067:L P[9125] 250mm/sec FINE;
1068:L P[9126] 250mm/sec CNT100;
1069:L P[9127] 250mm/sec CNT100;
1070:L P[9128] 250mm/sec FINE;
1071:L P[9129] 250mm/sec CNT100;
1072:L P[9130] 250mm/sec CNT100;
1073:L P[9131] 250mm/sec FINE;
1074:L P[9132] 250mm/sec CNT100;
1075:L P[9133] 250mm/sec CNT100;
1076:L P[9134] 250mm/sec FINE;
1077:L P[9135] 250mm/sec CNT100;
1078:L P[9136] 250mm/sec CNT100;
1079:L P[9137] 250mm/sec FINE;
1080:L P[9138] 250mm/sec CNT100;
1081:L P[9139] 250mm/sec CNT100;
1082:L P[9140] 250mm/sec FINE;
1083:L P[9141] 250mm/sec CNT100;
1084:L P[9142] 250mm/sec CNT100;
1085:L P[9143] 250mm/sec FINE;
1086:L P[9144] 250mm/sec CNT100;
1087:L P[9145] 250mm/sec CNT100;
1088:L P[9146] 250mm/sec FINE;
1089:L P[9147] 250mm/sec CNT100;
1090:L P[9148] 250mm/sec CNT100;
1091:L P[9149] 250mm/sec FINE;
1092:L P[9150] 250mm/sec CNT100;
1093:L P[9151] 250mm/sec CNT100;
1094:L P[9152] 250mm/sec FINE;
1095:L P[9153] 250mm/sec CNT100;
1096:L P[9154] 250mm/sec CNT100;
1097:L P[9155] 250mm/sec FINE;
1098:L P[9156] 250mm/sec CNT100;
1099:L P[9157] 250mm/sec CNT100;
1100:L P[9158] 250mm/sec FINE;
1101:L P[9159] 250mm/sec CNT100;
1102:L P[9160] 250mm/sec CNT100;
1103:L P[9161] 250mm/sec FINE;
1104:L P[9162] 250mm/sec CNT100;
1105:L P[9163] 250mm/sec CNT100;
1106:L P[9164] 250mm/sec FINE;
1107:L P[9165] 250mm/sec CNT100;
1108:L P[9166] 250mm/sec CNT100;
1109:L P[9167] 250mm/sec FINE;
1110:L P[9168] 250mm/sec CNT100;
1111:L P[9169] 250mm/sec CNT100;
1112:L P[9170] 250mm/sec FINE;
1113:L P[9171] 250mm/sec CNT100;
1114:L P[9172] 250mm/sec CNT100;
1115:L P[9173] 250mm/sec FINE;
1116:L P[9174] 250mm/sec CNT100;
1117:L P[9175] 250mm/sec CNT100;
1118:L P[9176] 250mm/sec FINE;
1119:L P[9177] 250mm/sec CNT100;
1120:L P[9178] 250mm/sec CNT100;
1121:L P[9179] 250mm/sec FINE;
1122:L P[9180] 250mm/sec CNT100;
1123:L P[9181] 250mm/sec CNT100;
1124:L P[9182] 250mm/sec FINE;
1125:L P[9183] 250mm/sec CNT100;
1126:L P[9184] 250mm/sec CNT100;
1127:L P[9185] 250mm/sec FINE;
1128:L P[9186] 250mm/sec CNT100;
1129:L P[9187] 250mm/sec CNT100;
1130:L P[9188] 250mm/sec FINE;
1131:L P[9189] 250mm/sec CNT100;
1132:L P[9190] 250mm/sec CNT100;
1133:L P[9191] 250mm/sec FINE;
1134:L P[9192] 250mm/sec CNT100;
1135:L P[9193] 250mm/sec CNT100;
1136:L P[9194] 250mm/sec FINE;
1137:L P[9195] 250mm/sec CNT100;
1138:L P[9196] 250mm/sec CNT100;
1139:L P[9197] 250mm/sec FINE;
1140:L P[9198] 250mm/sec CNT100;
1141:L P[9199] 250mm/sec CNT100;
1142:L P[9200] 250mm/sec FINE;
1143:L P[9201] 250mm/sec CNT100;
1144:L P[9202] 250mm/sec CNT100;
1145:L P[9203] 250mm/sec FINE;
1146:L P[9204] 250mm/sec CNT100;
1147:L P[9205] 250mm/sec CNT100;
1148:L P[9206] 250mm/sec FINE;
1149:L P[9207] 250mm/sec CNT100;
1150:L P[9208] 250mm/sec CNT100;
1151:L P[9209] 250mm/sec FINE;
1152:L P[9210] 250mm/sec CNT100;
1153:L P[9211] 250mm/sec CNT100;
1154:L P[9212] 250mm/sec FINE;
1155:L P[9213] 250mm/sec CNT100;
1156:L P[9214] 250mm/sec CNT100;
1157:L P[9215] 250mm/sec FINE;
1158:L P[9216] 250mm/sec CNT100;
1159:L P[9217] 250mm/sec CNT100;
1160:L P[9218] 250mm/sec FINE;
1161:L P[9219] 250mm/sec CNT100;
1162:L P[9220] 250mm/sec CNT100;
1163:L P[9221] 250mm/sec FINE;
1164:L P[9222] 250mm/sec CNT100;
1165:L P[9223] 250mm/sec CNT100;
1166:L P[9224] 250mm/sec FINE;
1167:L P[9225] 250mm/sec CNT100;
1168:L P[9226] 250mm/sec CNT100;
1169:L P[9227] 250mm/sec FINE;
1170:L P[9228] 250mm/sec CNT100;
1171:L P[9229] 250mm/sec CNT100;
1172:L P[9230] 250mm/sec FINE;
1173:L P[9231] 250mm/sec CNT100;
1174:L P[9232] 250mm/sec CNT100;
1175:L P[9233] 250mm/sec FINE;
1176:L P[9234] 250mm/sec CNT100;
1177:L P[9235] 250mm/sec CNT100;
1178:L P[9236] 250mm/sec FINE;
1179:L P[9237] 250mm/sec CNT100;
1180:L P[9238] 250mm/sec CNT100;
1181:L P[9239] 250mm/sec FINE;
1182:L P[9240] 250mm/sec CNT100;
1183:L P[9241] 250mm/sec CNT100;
1184:L P[9242] 250mm/sec FINE;
1185:L P[9243] 250mm/sec CNT100;
1186:L P[9244] 250mm/sec CNT100;
1187:L P[9245] 250mm/sec FINE;
1188:L P[9246] 250mm/sec CNT100;
1189:L P[9247] 250mm/sec CNT100;
1190:L P[9248] 250mm/sec FINE;
1191:L P[9249] 250mm/sec CNT100;
1192:L P[9250] 250mm/sec CNT100;
1193:L P[9251] 250mm/sec FINE;
1194:L P[9252] 250mm/sec CNT100;
1195:L P[9253] 250mm/sec CNT100;
1196:L P[9254] 250mm/sec FINE;
1197:L P[9255] 250mm/sec CNT100;
1198:L P[9256] 250mm/sec CNT100;
1199:L P[9257] 250mm/sec FINE;
1200:L P[9258] 250mm/sec CNT100;
1201:L P[9259] 250mm/sec CNT100;
1202:L P[9260] 250mm/sec FINE;
1203:L P[9261] 250mm/sec CNT100;
1204:L P[9262] 250mm/sec CNT100;
1205:L P[9263] 250mm/sec FINE;
1206:L P[9264] 250mm/sec CNT100;
1207:L P[9265] 250mm/sec CNT100;
1208:L P[9266] 250mm/sec FINE;
1209:L P[9267] 250mm/sec CNT100;
1210:L P[9268] 250mm/sec CNT100;
1211:L P[9269] 250mm/sec FINE;
1212:L P[9270] 250mm/sec CNT100;
1213:L P[9271] 250mm/sec CNT100;
1214:L P[9272] 250mm/sec FINE;
1215:L P[9273] 250mm/sec CNT100;
1216:L P[9274] 250mm/sec CNT100;
1217:L P[9275] 250mm/sec FINE;
1218:L P[9276] 250mm/sec CNT100;
1219:L P[9277] 250mm/sec CNT100;
1220:L P[9278] 250mm/sec FINE;
1221:L P[9279] 250mm/sec CNT100;
1222:L P[9280] 250mm/sec CNT100;
1223:L P[9281] 250mm/sec FINE;
1224:L P[9282] 250mm/sec CNT100;
1225:L P[9283] 250mm/sec CNT100;
1226:L P[9284] 250mm/sec FINE;
1227:L P[9285] 250mm/sec CNT100;
1228:L P[9286] 250mm/sec CNT100;
1229:L P[9287] 250mm/sec FINE;
1230:L P[9288] 250mm/sec CNT100;
1231:L P[9289] 250mm/sec CNT100;
1232:L P[9290] 250mm/sec FINE;
1233:L P[9291] 250mm/sec CNT100;
1234:L P[9292] 250mm/sec CNT100;
1235:L P[9293] 250mm/sec FINE;
1236:L P[9294] 250mm/sec CNT100;
1237:L P[9295] 250mm/sec CNT100;
1238:L P[9296] 250mm/sec FINE;
1239:L P[9297] 250mm/sec CNT100;
1240:L P[9298] 250mm/sec CNT100;
1241:L P[9299] 250mm/sec FINE;
1242:L P[9300] 250mm/sec CNT100;
1243:L P[9301] 250mm/sec CNT100;
1244:L P[9302] 250mm/sec FINE;
1245:L P[9303] 250mm/sec CNT100;
1246:L P[9304] 250mm/sec CNT100;
1247:L P[9305] 250mm/sec FINE;
1248:L P[9306] 250mm/sec CNT100;
1249:L P[9307] 250mm/sec CNT100;
1250:L P[9308] 250mm/sec FINE;
1251:L P[9309] 250mm/sec CNT100;
1252:L P[9310] 250mm/sec CNT100;
1253:L P[9311] 250mm/sec FINE;
1254:L P[9312] 250mm/sec CNT100;
1255:L P[9313] 250mm/sec CNT100;
1256:L P[9314] 250mm/sec FINE;
1257:L P[9315] 250mm/sec CNT100;
1258:L P[9316] 250mm/sec CNT100;
1259:L P[9317] 250mm/sec FINE;
1260:L P[9318] 250mm/sec CNT100;
1261:L P[9319] 250mm/sec CNT100;
1262:L P[9320] 250mm/sec FINE;
1263:L P[9321] 250mm/sec CNT100;
1264:L P[9322] 250mm/sec CNT100;
1265:L P[9323] 250mm/sec FINE;
1266:L P[9324] 250mm/sec CNT100;
1267:L P[9325] 250mm/sec CNT100;
1268:L P[9326] 250mm/sec FINE;
1269:L P[9327] 250mm/sec CNT100;
1270:L P[9328] 250mm/sec CNT100;
1271:L P[9329] 250mm/sec FINE;
1272:L P[9330] 250mm/sec CNT100;
1273:L P[9331] 250mm/sec CNT100;
1274:L P[9332] 250mm/sec FINE;
1275:L P[9333] 250mm/sec CNT100;
1276:L P[9334] 250mm/sec CNT100;
1277:L P[9335] 250mm/sec FINE;
1278:L P[9336] 250mm/sec CNT100;
1279:L P[9337] 250mm/sec CNT100;
1280:L P[9338] 250mm/sec FINE;
1281:L P[9339] 250mm/sec CNT100;
1282:L P[9340] 250mm/sec CNT100;
1283:L P[9341] 250mm/sec FINE;
1284:L P[9342] 250mm/sec CNT100;
1285:L P[9343] 250mm/sec CNT100;
1286:L P[9344] 250mm/sec FINE;
1287:L P[9345] 250mm/sec CNT100;
1288:L P[9346] 250mm/sec CNT100;
1289:L P[9347] 250mm/sec FINE;
1290:L P[9348] 250mm/sec CNT100;
1291:L P[9349] 250mm/sec CNT100;
1292:L P[9350] 250mm/sec FINE;
1293:L P[9351] 250mm/sec CNT100;
1294:L P[9352] 250mm/sec CNT100;
1295:L P[9353] 250mm/sec FINE;
1296:L P[9354] 250mm/sec CNT100;
1297:L P[9355] 250mm/sec CNT100;
1298:L P[9356] 250mm/sec FINE;
1299:L P[9357] 250mm/sec CNT100;
1300:L P[9358] 250mm/sec CNT100;
1301:L P[9359] 250mm/sec FINE;
1302:L P[9360] 250mm/sec CNT100;
1303:L P[9361] 250mm/sec CNT100;
1304:L P[9362] 250mm/sec FINE;
1305:L P[9363] 250mm/sec CNT100;
1306:L P[9364] 250mm/sec CNT100;
1307:L P[9365] 250mm/sec FINE;
1308:L P[9366] 250mm/sec CNT100;
1309:L P[9367] 250mm/sec CNT100;
1310:L P[9368] 250mm/sec FINE;
1311:L P[9369] 250mm/sec CNT100;
1312:L P[9370] 250mm/sec CNT100;
1313:L P[9371] 250mm/sec FINE;
1314:L P[9372] 250mm/sec CNT100;
1315:L P[9373] 250mm/sec CNT100;
1316:L P[9374] 250mm/sec FINE;
1317:L P[9375] 250mm/sec CNT100;
1318:L P[9376] 250mm/sec CNT100;
1319:L P[9377] 250mm/sec FINE;
1320:L P[9378] 250mm/sec CNT100;
1321:L P[9379] 250mm/sec CNT100;
1322:L P[9380] 250mm/sec FINE;
1323:L P[9381] 250mm/sec CNT100;
1324:L P[9382] 250mm/sec CNT100;
1325:L P[9383] 250mm/sec FINE;
1326:L P[9384] 250mm/sec CNT100;
1327:L P[9385] 250mm/sec CNT100;
1328:L P[9386] 250mm/sec FINE;
1329:L P[9387] 250mm/sec CNT100;
1330:L P[9388] 250mm/sec CNT100;
1331:L P[9389] 250mm/sec FINE;
1332:L P[9390] 250mm/sec CNT100;
1333:L P[9391] 250mm/sec CNT100;
1334:L P[9392] 250mm/sec FINE;
1335:L P[9393] 250mm/sec CNT100;
1336:L P[9394] 250mm/sec CNT100;
1337:L P[9395] 250mm/sec FINE;
1338:L P[9396] 250mm/sec CNT100;
1339:L P[9397] 250mm/sec CNT100;
1340:L P[9398] 250mm/sec FINE;
1341:L P[9399] 250mm/sec CNT100;
1342:L P[9400] 250mm/sec CNT100;
1343:L P[9401] 250mm/sec FINE;
1344:L P[9402] 250mm/sec CNT100;
1345:L P[9403] 250mm/sec CNT100;
1346:L P[9404] 250mm/sec FINE;
1347:L P[9405] 250mm/sec CNT100;
1348:L P[9406] 250mm/sec CNT100;
1349:L P[9407] 250mm/sec FINE;
1350:L P[9408] 250mm/sec CNT100;
1351:L P[9409] 250mm/sec CNT100;
1352:L P[9410] 250mm/sec FINE;
1353:L P[9411] 250mm/sec CNT100;
1354:L P[9412] 250mm/sec CNT100;
1355:L P[9413] 250mm/sec FINE;
1356:L P[9414] 250mm/sec CNT100;
1357:L P[9415] 250mm/sec CNT100;
1358:L P[9416] 250mm/sec FINE;
1359:L P[9417] 250mm/sec CNT100;
1360:L P[9418] 250mm/sec CNT100;
1361:L P[9419] 250mm/sec FINE;
1362:L P[9420] 250mm/sec CNT100;
1363:L P[9421] 250mm/sec CNT100;
1364:L P[9422] 250mm/sec FINE;
1365:L P[9423] 250mm/sec CNT100;
1366:L P[9424] 250mm/sec CNT100;
1367:L P[9425] 250mm/sec FINE;
1368:L P[9426] 250mm/sec CNT100;
1369:L P[9427] 250mm/sec CNT100;
1370:L P[9428] 250mm/sec FINE;
1371:L P[9429] 250mm/sec CNT100;
1372:L P[9430] 250mm/sec CNT100;
1373:L P[9431] 250mm/sec FINE;
1374:L P[9432] 250mm/sec CNT100;
1375:L P[9433] 250mm/sec CNT100;
1376:L P[9434] 250mm/sec FINE;
1377:L P[9435] 250mm/sec CNT100;
1378:L P[9436] 250mm/sec CNT100;
1379:L P[9437] 250mm/sec FINE;
1380:L P[9438] 250mm/sec CNT100;
1381:L P[9439] 250mm/sec CNT100;
1382:L P[9440] 250mm/sec FINE;
1383:L P[9441] 250mm/sec CNT100;
1384:L P[9442] 250mm/sec CNT100;
1385:L P[9443] 250mm/sec FINE;
1386:L P[9444] 250mm/sec CNT100;
1387:L P[9445] 250mm/sec CNT100;
1388:L P[9446] 250mm/sec FINE;
1389:L P[9447] 250mm/sec CNT100;
1390:L P[9448] 250mm/sec CNT100;
1391:L P[9449] 250mm/sec FINE;
1392:L P[9450] 250mm/sec CNT100;
1393:L P[9451] 250mm/sec CNT100;
1394:L P[9452] 250mm/sec FINE;
1395:L P[9453] 250mm/sec CNT100;
1396:L P[9454] 250mm/sec CNT100;
1397:L P[9455] 250mm/sec FINE;
1398:L P[9456] 250mm/sec CNT100;
1399:L P[9457] 250mm/sec CNT100;
1400:L P[9458] 250mm/sec FINE;
1401:L P[9459] 250mm/sec CNT100;
1402:L P[9460] 250mm/sec CNT100;
1403:L P[9461] 250mm/sec FINE;
1404:L P[9462] 250mm/sec CNT100;
1405:L P[9463] 250mm/sec CNT100;
1406:L P[9464] 250mm/sec FINE;
1407:L P[9465] 250mm/sec CNT100;
1408:L P[9466] 250mm/sec CNT100;
1409:L P[9467] 250mm/sec FINE;
1410:L P[9468] 250mm/sec CNT100;
1411:L P[9469] 250mm/sec CNT100;
1412:L P[9470] 250mm/sec FINE;
1413:L P[9471] 250mm/sec CNT100;
1414:L P[9472] 250mm/sec CNT100;
1415:L P[9473] 250mm/sec FINE;
1416:L P[9474] 250mm/sec CNT100;
1417:L P[9475] 250mm/sec CNT100;
1418:L P[9476] 250mm/sec FINE;
1419:L P[9477] 250mm/sec CNT100;
1420:L P[9478] 250mm/sec CNT100;
1421:L P[9479] 250mm/sec FINE;
1422:L P[9480] 250mm/sec CNT100;
1423:L P[9481] 250mm/sec CNT100;
1424:L P[9482] 250mm/sec FINE;
1425:L P[9483] 250mm/sec CNT100;
1426:L P[9484] 250mm/sec CNT100;
1427:L P[9485] 250mm/sec FINE;
1428:L P[9486] 250mm/sec CNT100;
1429:L P[9487] 250mm/sec CNT100;
1430:L P[9488] 250mm/sec FINE;
1431:L P[9489] 250mm/sec CNT100;
1432:L P[9490] 250mm/sec CNT100;
1433:L P[9491] 250mm/sec FINE;
1434:L P[9492] 250mm/sec CNT100;
1435:L P[9493] 250mm/sec CNT100;
1436:L P[9494] 250mm/sec FINE;
1437:L P[9495] 250mm/sec CNT100;
1438:L P[9496] 250mm/sec CNT100;
1439:L P[9497] 250mm/sec FINE;
1440:L P[9498] 250mm/sec CNT100;
1441:L P[9499] 250mm/sec CNT100;
1442:L P[9500] 250mm/sec FINE;
1443:L P[9501] 250mm/sec CNT100;
1444:L P[9502] 250mm/sec CNT100;
1445:L P[9503] 250mm/sec FINE;
1446:L P[9504] 250mm/sec CNT100;
1447:L P[9505] 250mm/sec CNT100;
1448:L P[9506] 250mm/sec FINE;
1449:L P[9507] 250mm/sec CNT100;
1450:L P[9508] 250mm/sec CNT100;
1451:L P[9509] 250mm/sec FINE;
1452:L P[9510] 250mm/sec CNT100;
1453:L P[9511] 250mm/sec CNT100;
1454:L P[9512] 250mm/sec FINE;
1455:L P[9513] 250mm/sec CNT100;
1456:L P[9514] 250mm/sec CNT100;
1457:L P[9515] 250mm/sec FINE;
1458:L P[9516] 250mm/sec CNT100;
1459:L P[9517] 250mm/sec CNT100;
1460:L P[9518] 250mm/sec FINE;
1461:L P[9519] 250mm/sec CNT100;
1462:L P[9520] 250mm/sec CNT100;
1463:L P[9521] 250mm/sec FINE;
1464:L P[9522] 250mm/sec CNT100;
1465:L P[9523] 250mm/sec CNT100;
1466:L P[9524] 250mm/sec FINE;
1467:L P[9525] 250mm/sec CNT100;
1468:L P[9526] 250mm/sec CNT100;
1469:L P[9527] 250mm/sec FINE;
1470:L P[9528] 250mm/sec CNT100;
1471:L P[9529] 250mm/sec CNT100;
1472:L P[9530] 250mm/sec FINE;
1473:L P[9531] 250mm/sec CNT100;
1474:L P[9532] 250mm/sec CNT100;
1475:L P[9533] 250mm/sec FINE;
1476:L P[9534] 250mm/sec CNT100;
1477:L P[9535] 250mm/sec CNT100;
1478:L P[9536] 250mm/sec FINE;
1479:L P[9537] 250mm/sec CNT100;
1480:L P[9538] 250mm/sec CNT100;
1481:L P[9539] 250mm/sec FINE;
1482:L P[9540] 250mm/sec CNT100;
1483:L P[9541] 250mm/sec CNT100;
1484:L P[9542] 250mm/sec FINE;
1485:L P[9543] 250mm/sec CNT100;
1486:L P[9544] 250mm/sec CNT100;
1487:L P[9545] 250mm/sec FINE;
1488:L P[9546] 250mm/sec CNT100;
1489:L P[9547] 250mm/sec CNT100;
1490:L P[9548] 250mm/sec FINE;
1491:L P[9549] 250mm/sec CNT100;
1492:L P[9550] 250mm/sec CNT100;
1493:L P[9551] 250mm/sec FINE;
1494:L P[9552] 250mm/sec CNT100;
1495:L P[9553] 250mm/sec CNT100;
1496:L P[9554] 250mm/sec FINE;
1497:L P[9555] 250mm/sec CNT100;
1498:L P[9556] 250mm/sec CNT100;
1499:L P[9557] 250mm/sec FINE;
1500:L P[9558] 250mm/sec CNT100;
1501:L P[9559] 250mm/sec CNT100;
1502:L P[9560] 250mm/sec FINE;
1503:L P[9561] 250mm/sec CNT100;
1504:L P[9562] 250mm/sec CNT100;
1505:L P[9563] 250mm/sec FINE;
1506:L P[9564] 250mm/sec CNT100;
1507:L P[9565] 250mm/sec CNT100;
1508:L P[9566] 250mm/sec FINE;
1509:L P[9567] 250mm/sec CNT100;
1510:L P[9568] 250mm/sec CNT100;
1511:L P[9569] 250mm/sec FINE;
1512:L P[9570] 250mm/sec CNT100;
1513:L P[9571] 250mm/sec CNT100;
1514:L P[9572] 250mm/sec FINE;
1515:L P[9573] 250mm/sec CNT100;
1516:L P[9574] 250mm/sec CNT100;
1517:L P[9575] 250mm/sec FINE;
1518:L P[9576] 250mm/sec CNT100;
1519:L P[9577] 250mm/sec CNT100;
1520:L P[9578] 250mm/sec FINE;
1521:L P[9579] 250mm/sec CNT100;
1522:L P[9580] 250mm/sec CNT100;
1523:L P[9581] 250mm/sec FINE;
1524:L P[9582] 250mm/sec CNT100;
1525:L P[9583] 250mm/sec CNT100;
1526:L P[9584] 250mm/sec FINE;
1527:L P[9585] 250mm/sec CNT100;
1528:L P[9586] 250mm/sec CNT100;
1529:L P[9587] 250mm/sec FINE;
1530:L P[9588] 250mm/sec CNT100;
1531:L P[9589] 250mm/sec CNT100;
1532:L P[9590] 250mm/sec FINE;
1533:L P[9591] 250mm/sec CNT100;
1534:L P[9592] 250mm/sec CNT100;
1535:L P[9593] 250mm/sec FINE;
1536:L P[9594] 250mm/sec CNT100;
1537:L P[9595] 250mm/sec CNT100;
1538:L P[9596] 250mm/sec FINE;
1539:L P[9597] 250mm/sec CNT100;
1540:L P[9598] 250mm/sec CNT100;
1541:L P[9599] 250mm/sec FINE;
1542:L P[9600] 250mm/sec CNT100;
1543:L P[9601] 250mm/sec CNT100;
1544:L P[9602] 250mm/sec FINE;
1545:L P[9603] 250mm/sec CNT100;
1546:L P[9604] 250mm/sec CNT100;
1547:L P[9605] 250mm/sec FINE;
1548:L P[9606] 250mm/sec CNT100;
1549:L P[9607] 250mm/sec CNT100;
1550:L P[9608] 250mm/sec FINE;
1551:L P[9609] 250mm/sec CNT100;
1552:L P[9610] 250mm/sec CNT100;
1553:L P[9611] 250mm/sec FINE;
1554:L P[9612] 250mm/sec CNT100;
1555:L P[9613] 250mm/sec CNT100;
1556:L P[9614] 250mm/sec FINE;
1557:L P[9615] 250mm/sec CNT100;
1558:L P[9616] 250mm/sec CNT100;
1559:L P[9617] 250mm/sec FINE;
1560:L P[9618] 250mm/sec CNT100;
1561:L P[9619] 250mm/sec CNT100;
1562:L P[9620] 250mm/sec FINE;
1563:L P[9621] 250mm/sec CNT100;
1564:L P[9622] 250mm/sec CNT100;
1565:L P[9623] 250mm/sec FINE;
1566:L P[9624] 250mm/sec CNT100;
1567:L P[9625] 250mm/sec CNT100;
1568:L P[9626] 250mm/sec FINE;
1569:L P[9627] 250mm/sec CNT100;
1570:L P[9628] 250mm/sec CNT100;
1571:L P[9629] 250mm/sec FINE;
1572:L P[9630] 250mm/sec CNT100;
1573:L P[9631] 250mm/sec CNT100;
1574:L P[9632] 250mm/sec FINE;
1575:L P[9633] 250mm/sec CNT100;
1576:L P[9634] 250mm/sec CNT100;
1577:L P[9635] 250mm/sec FINE;
1578:L P[9636] 250mm/sec CNT100;
1579:L P[9637] 250mm/sec CNT100;
1580:L P[9638] 250mm/sec FINE;
1581:L P[9639] 250mm/sec CNT100;
1582:L P[9640] 250mm/sec CNT100;
1583:L P[9641] 250mm/sec FINE;
1584:L P[9642] 250mm/sec CNT100;
1585:L P[9643] 250mm/sec CNT100;
1586:L P[9644] 250mm/sec FINE;
1587:L P[9645] 250mm/sec CNT100;
1588:L P[9646] 250mm/sec CNT100;
1589:L P[9647] 250mm/sec FINE;
1590:L P[9648] 250mm/sec CNT100;
1591:L P[9649] 250mm/sec CNT100;
1592:L P[9650] 250mm/sec FINE;
1593:L P[9651] 250mm/sec CNT100;
1594:L P[9652] 250mm/sec CNT100;
1595:L P[9653] 250mm/sec FINE;
1596:L P[9654] 250mm/sec CNT100;
1597:L P[9655] 250mm/sec CNT100;
1598:L P[9656] 250mm/sec FINE;
1599:L P[9657] 250mm/sec CNT100;
1600:L P[9658] 250mm/sec CNT100;
1601:L P[9659] 250mm/sec FINE;
1602:L P[9660] 250mm/sec CNT100;
1603:L P[9661] 250mm/sec CNT100;
1604:L P[9662] 250mm/sec FINE;
1605:L P[9663] 250mm/sec CNT100;
1606:L P[9664] 250mm/sec CNT100;
1607:L P[9665] 250mm/sec FINE;
1608:L P[9666] 250mm/sec CNT100;
1609:L P[9667] 250mm/sec CNT100;
1610:L P[9668] 250mm/sec FINE;
1611:L P[9669] 250mm/sec CNT100;
1612:L P[9670] 250mm/sec CNT100;
1613:L P[9671] 250mm/sec FINE;
1614:L P[9672] 250mm/sec CNT100;
1615:L P[9673] 250mm/sec CNT100;
1616:L P[9674] 250mm/sec FINE;
1617:L P[9675] 250mm/sec CNT100;
1618:L P[9676] 250mm/sec CNT100;
1619:L P[9677] 250mm/sec FINE;
1620:L P[9678] 250mm/sec CNT100;
1621:L P[9679] 250mm/sec CNT100;
1622:L P[9680] 250mm/sec FINE;
1623:L P[9681] 250mm/sec CNT100;
1624:L P[9682] 250mm/sec CNT100;
1625:L P[9683] 250mm/sec FINE;
1626:L P[9684] 250mm/sec CNT100;
1627:L P[9685] 250mm/sec CNT100;
1628:L P[9686] 250mm/sec FINE;
1629:L P[9687] 250mm/sec CNT100;
1630:L P[9688] 250mm/sec CNT100;
1631:L P[9689] 250mm/sec FINE;
1632:L P[9690] 250mm/sec CNT100;
1633:L P[9691] 250mm/sec CNT100;
1634:L P[9692] 250mm/sec FINE;
1635:L P[9693] 250mm/sec CNT100;
1636:L P[9694] 250mm/sec CNT100;
1637:L P[9695] 250mm/sec FINE;
1638:L P[9696] 250mm/sec CNT100;
1639:L P[9697] 250mm/sec CNT100;
1640:L P[9698] 250mm/sec FINE;
1641:L P[9699] 250mm/sec CNT100;
1642:L P[9700] 250mm/sec CNT100;
1643:L P[9701] 250mm/sec FINE;
1644:L P[9702] 250mm/sec CNT100;
1645:L P[9703] 250mm/sec CNT100;
1646:L P[9704] 250mm/sec FINE;
1647:L P[9705] 250mm/sec CNT100;
1648:L P[9706] 250mm/sec CNT100;
1649:L P[9707] 250mm/sec FINE;
1650:L P[9708] 250mm/sec CNT100;
1651:L P[9709] 250mm/sec CNT100;
1652:L P[9710] 250mm/sec FINE;
1653:L P[9711] 250mm/sec CNT100;
1654:L P[9712] 250mm/sec CNT100;
1655:L P[9713] 250mm/sec FINE;
1656:L P[9714] 250mm/sec CNT100;
1657:L P[9715] 250mm/sec CNT100;
1658:L P[9716] 250mm/sec FINE;
1659:L P[9717] 250mm/sec CNT100;
1660:L P[9718] 250mm/sec CNT100;
1661:L P[9719] 250mm/sec FINE;
1662:L P[9720] 250mm/sec CNT100;
1663:L P[9721] 250mm/sec CNT100;
1664:L P[9722] 250mm/sec FINE;
1665:L P[9723] 250mm/sec CNT100;
1666:L P[9724] 250mm/sec CNT100;
1667:L P[9725] 250mm/sec FINE;
1668:L P[9726] 250mm/sec CNT100;
1669:L P[9727] 250mm/sec CNT100;
1670:L P[9728] 250mm/sec FINE;
1671:L P[9729] 250mm/sec CNT100;
1672:L P[9730] 250mm/sec CNT100;
1673:L P[9731] 250mm/sec FINE;
1674:L P[9732] 250mm/sec CNT100;
1675:L P[9733] 250mm/sec CNT100;
1676:L P[9734] 250mm/sec FINE;
1677:L P[9735] 250mm/sec CNT100;
1678:L P[9736] 250mm/sec CNT100;
1679:L P[9737] 250mm/sec FINE;
1680:L P[9738] 250mm/sec CNT100;
1681:L P[9739] 250mm/sec CNT100;
1682:L P[9740] 250mm/sec FINE;
1683:L P[9741] 250mm/sec CNT100;
1684:L P[9742] 250mm/sec CNT100;
1685:L P[9743] 250mm/sec FINE;
1686:L P[9744] 250mm/sec CNT100;
1687:L P[9745] 250mm/sec CNT100;
1688:L P[9746] 250mm/sec FINE;
1689:L P[9747] 250mm/sec CNT100;
1690:L P[9748] 250mm/sec CNT100;
1691:L P[9749] 250mm/sec FINE;
1692:L P[9750] 250mm/sec CNT100;
1693:L P[9751] 250mm/sec CNT100;
1694:L P[9752] 250mm/sec FINE;
1695:L P[9753] 250mm/sec CNT100;
1696:L P[9754] 250mm/sec CNT100;
1697:L P[9755] 250mm/sec FINE;
1698:L P[9756] 250mm/sec CNT100;
1699:L P[9757] 250mm/sec CNT100;
1700:L P[9758] 250mm/sec FINE;
1701:L P[9759] 250mm/sec CNT100;
1702:L P[9760] 250mm/sec CNT100;
1703:L P[9761] 250mm/sec FINE;
1704:L P[9762] 250mm/sec CNT100;
1705:L P[9763] 250mm/sec CNT100;
1706:L P[9764] 250mm/sec FINE;
1707:L P[9765] 250mm/sec CNT100;
1708:L P[9766] 250mm/sec CNT100;
1709:L P[9767] 250mm/sec FINE;
1710:L P[9768] 250mm/sec CNT100;
1711:L P[9769] 250mm/sec CNT100;
1712:L P[9770] 250mm/sec FINE;
1713:L P[9771] 250mm/sec CNT100;
1714:L P[9772] 250mm/sec CNT100;
1715:L P[9773] 250mm/sec FINE;
1716:L P[9774] 250mm/sec CNT100;
1717:L P[9775] 250mm/sec CNT100;
1718:L P[9776] 250mm/sec FINE;
1719:L P[9777] 250mm/sec CNT100;
1720:L P[9778] 250mm/sec CNT100;
1721:L P[9779] 250mm/sec FINE;
1722:L P[9780] 250mm/sec CNT100;
1723:L P[9781] 250mm/sec CNT100;
1724:L P[9782] 250mm/sec FINE;
1725:L P[9783] 250mm/sec CNT100;
1726:L P[9784] 250mm/sec CNT100;
1727:L P[9785] 250mm/sec FINE;
1728:L P[9786] 250mm/sec CNT100;
1729:L P[9787] 250mm/sec CNT100;
1730:L P[9788] 250mm/sec FINE;
1731:L P[9789] 250mm/sec CNT100;
1732:L P[9790] 250mm/sec CNT100;
1733:L P[9791] 250mm/sec FINE;
1734:L P[9792] 250mm/sec CNT100;
1735:L P[9793] 250mm/sec CNT100;
1736:L P[9794] 250mm/sec FINE;
1737:L P[9795] 250mm/sec CNT100;
1738:L P[9796] 250mm/sec CNT100;
1739:L P[9797] 250mm/sec FINE;
1740:L P[9798] 250mm/sec CNT100;
1741:L P[9799] 250mm/sec CNT100;
1742:L P[9800] 250mm/sec FINE;
1743:L P[9801] 250mm/sec CNT100;
1744:L P[9802] 250mm/sec CNT100;
1745:L P[9803] 250mm/sec FINE;
1746:L P[9804] 250mm/sec CNT100;
1747:L P[9805] 250mm/sec CNT100;
1748:L P[9806] 250mm/sec FINE;
1749:L P[9807] 250mm/sec CNT100;
1750:L P[9808] 250mm/sec CNT100;
1751:L P[9809] 250mm/sec FINE;
1752:L P[9810] 250mm/sec CNT100;
1753:L P[9811] 250mm/sec CNT100;
1754:L P[9812] 250mm/sec FINE;
1755:L P[9813] 250mm/sec CNT100;
1756:L P[9814] 250mm/sec CNT100;
1757:L P[9815] 250mm/sec FINE;
1758:L P[9816] 250mm/sec CNT100;
1759:L P[9817] 250mm/sec CNT100;
1760:L P[9818] 250mm/sec FINE;
1761:L P[9819] 250mm/sec CNT100;
1762:L P[9820] 250mm/sec CNT100;
1763:L P[9821] 250mm/sec FINE;
1764:L P[9822] 250mm/sec CNT100;
1765:L P[9823] 250mm/sec CNT100;
1766:L P[9824] 250mm/sec FINE;
1767:L P[9825] 250mm/sec CNT100;
1768:L P[9826] 250mm/sec CNT100;
1769:L P[9827] 250mm/sec FINE;
1770:L P[9828] 250mm/sec CNT100;
1771:L P[9829] 250mm/sec CNT100;
1772:L P[9830] 250mm/sec FINE;
1773:L P[9831] 250mm/sec CNT100;
1774:L P[9832] 250mm/sec CNT100;
1775:L P[9833] 250mm/sec FINE;
1776:L P[9834] 250mm/sec CNT100;
1777:L P[9835] 250mm/sec CNT100;
1778:L P[9836] 250mm/sec FINE;
1779:L P[9837] 250mm/sec CNT100;
1780:L P[9838] 250mm/sec CNT100;
1781:L P[9839] 250mm/sec FINE;
1782:L P[9840] 250mm/sec CNT100;
1783:L P[9841] 250mm/sec CNT100;
1784:L P[9842] 250mm/sec FINE;
1785:L P[9843] 250mm/sec CNT100;
1786:L P[9844] 250mm/sec CNT100;
1787:L P[9845] 250mm/sec FINE;
1788:L P[9846] 250mm/sec CNT100;
1789:L P[9847] 250mm/sec CNT100;
1790:L P[9848] 250mm/sec FINE;
1791:L P[9849] 250mm/sec CNT100;
1792:L P[9850] 250mm/sec CNT100;
1793:L P[9851] 250mm/sec FINE;
1794:L P[9852] 250mm/sec CNT100;
1795:L P[9853] 250mm/sec CNT100;
1796:L P[9854] 250mm/sec FINE;
1797:L P[9855] 250mm/sec CNT100;
1798:L P[9856] 250mm/sec CNT100;
1799:L P[9857] 250mm/sec FINE;
1800:L P[9858] 250mm/sec CNT100;
1801:L P[9859] 250mm/sec CNT100;
1802:L P[9860] 250mm/sec FINE;
1803:L P[9861] 250mm/sec CNT100;
1804:L P[9862] 250mm/sec CNT100;
1805:L P[9863] 250mm/sec FINE;
1806:L P[9864] 250mm/sec CNT100;
1807:L P[9865] 250mm/sec CNT100;
1808:L P[9866] 250mm/sec FINE;
1809:L P[9867] 250mm/sec CNT100;
1810:L P[9868] 250mm/sec CNT100;
1811:L P[9869] 250mm/sec FINE;
1812:L P[9870] 250mm/sec CNT100;
1813:L P[9871] 250mm/sec CNT100;
1814:L P[9872] 250mm/sec FINE;
1815:L P[9873] 250mm/sec CNT100;
1816:L P[9874] 250mm/sec CNT100;
1817:L P[9875] 250mm/sec FINE;
1818:L P[9876] 250mm/sec CNT100;
1819:L P[9877] 250mm/sec CNT100;
1820:L P[9878] 250mm/sec FINE;
1821:L P[9879] 250mm/sec CNT100;
1822:L P[9880] 250mm/sec CNT100;
1823:L P[9881] 250mm/sec FINE;
1824:L P[9882] 250mm/sec CNT100;
1825:L P[9883] 250mm/sec CNT100;
1826:L P[9884] 250mm/sec FINE;
1827:L P[9885] 250mm/sec CNT100;
1828:L P[9886] 250mm/sec CNT100;
1829:L P[9887] 250mm/sec FINE;
1830:L P[9888] 250mm/sec CNT100;
1831:L P[9889] 250mm/sec CNT100;
1832:L P[9890] 250mm/sec FINE;
1833:L P[9891] 250mm/sec CNT100;
1834:L P[9892] 250mm/sec CNT100;
1835:L P[9893] 250mm/sec FINE;
1836:L P[9894] 250mm/sec CNT100;
1837:L P[9895] 250mm/sec CNT100;
1838:L P[9896] 250mm/sec FINE;
1839:L P[9897] 250mm/sec CNT100;
1840:L P[9898] 250mm/sec CNT100;
1841:L P[9899] 250mm/sec FINE;
1842:L P[9900] 250mm/sec CNT100;
1843:L P[9901] 250mm/sec CNT100;
1844:L P[9902] 250mm/sec FINE;
1845:L P[9903] 250mm/sec CNT100;
1846:L P[9904] 250mm/sec CNT100;
1847:L P[9905] 250mm/sec FINE;
1848:L P[9906] 250mm/sec CNT100;
1849:L P[9907] 250mm/sec CNT100;
1850:L P[9908] 250mm/sec FINE;
1851:L P[9909] 250mm/sec CNT100;
1852:L P[9910] 250mm/sec CNT100;
1853:L P[9911] 250mm/sec FINE;
1854:L P[9912] 250mm/sec CNT100;
1855:L P[9913] 250mm/sec CNT100;
1856:L P[9914] 250mm/sec FINE;
1857:L P[9915] 250mm/sec CNT100;
1858:L P[9916] 250mm/sec CNT100;
1859:L P[9917] 250mm/sec FINE;
1860:L P[9918] 250mm/sec CNT100;
1861:L P[9919] 250mm/sec CNT100;
1862:L P[9920] 250mm/sec FINE;
1863:L P[9921] 250mm/sec CNT100;
1864:L P[9922] 250mm/sec CNT100;
1865:L P[9923] 250mm/sec FINE;
1866:L P[9924] 250mm/sec CNT100;
1867:L P[9925] 250mm/sec CNT100;
1868:L P[9926] 250mm/sec FINE;
1869:L P[9927] 250mm/sec CNT100;
1870:L P[9928] 250mm/sec CNT100;
1871:L P[9929] 250mm/sec FINE;
1872:L P[9930] 250mm/sec CNT100;
1873:L P[9931] 250mm/sec CNT100;
1874:L P[9932] 250mm/sec FINE;
1875:L P[9933] 250mm/sec CNT100;
1876:L P[9934] 250mm/sec CNT100;
1877:L P[9935] 250mm/sec FINE;
1878:L P[9936] 250mm/sec CNT100;
1879:L P[9937] 250mm/sec CNT100;
1880:L P[9938] 250mm/sec FINE;
1881:L P[9939] 250mm/sec CNT100;
1882:L P[9940] 250mm/sec CNT100;
1883:L P[9941] 250mm/sec FINE;
1884:L P[9942] 250mm/sec CNT100;
1885:L P[9943] 250mm/sec CNT100;
1886:L P[9944] 250mm/sec FINE;
1887:L P[9945] 250mm/sec CNT100;
1888:L P[9946] 250mm/sec CNT100;
1889:L P[9947] 250mm/sec FINE;
1890:L P[9948] 250mm/sec CNT100;
1891:L P[9949] 250mm/sec CNT100;
1892:L P[9950] 250mm/sec FINE;
1893:L P[9951] 250mm/sec CNT100;
1894:L P[9952] 250mm/sec CNT100;
1895:L P[9953] 250mm/sec FINE;
1896:L P[9954] 250mm/sec CNT100;
1897:L P[9955] 250mm/sec CNT100;
1898:L P[9956] 250mm/sec FINE;
1899:L P[9957] 250mm/sec CNT100;
1900:L P[9958] 250mm/sec CNT100;
1901:L P[9959] 250mm/sec FINE;
1902:L P[9960] 250mm/sec CNT100;
1903:L P[9961] 250mm/sec CNT100;
1904:L P[9962] 250mm/sec FINE;
1905:L P[9963] 250mm/sec CNT100;
1906:L P[9964] 250mm/sec CNT100;
1907:L P[9965] 250mm/sec FINE;
1908:L P[9966] 250mm/sec CNT100;
1909:L P[9967] 250mm/sec CNT100;
1910:L P[9968] 250mm/sec FINE;
1911:L P[9969] 250mm/sec CNT100;
1912:L P[9970] 250mm/sec CNT100;
1913:L P[9971] 250mm/sec FINE;
1914:L P[9972] 250mm/sec CNT100;
1915:L P[9973] 250mm/sec CNT100;
1916:L P[9974] 250mm/sec FINE;
1917:L P[9975] 250mm/sec CNT100;
1918:L P[9976] 250mm/sec CNT100;
1919:L P[9977] 250mm/sec FINE;
1920:L P[9978] 250mm/sec CNT100;
1921:L P[9979] 250mm/sec CNT100;
1922:L P[9980] 250mm/sec FINE;
1923:L P[9981] 250mm/sec CNT100;
1924:L P[9982] 250mm/sec CNT100;
1925:L P[9983] 250mm/sec FINE;
1926:L P[9984] 250mm/sec CNT100;
1927:L P[9985] 250mm/sec CNT100;
1928:L P[9986] 250mm/sec FINE;
1929:L P[9987] 250mm/sec CNT100;
1930:L P[9988] 250mm/sec CNT100;
1931:L P[9989] 250mm/sec FINE;
1932:L P[9990] 250mm/sec CNT100;
1933:L P[9991] 250mm/sec CNT100;
1934:L P[9992] 250mm/sec FINE;
1935:L P[9993] 250mm/sec CNT100;
1936:L P[9994] 250mm/sec CNT100;
1937:L P[9995] 250mm/sec FINE;
1938:L P[9996] 250mm/sec CNT100;
1939:L P[9997] 250mm/sec CNT100;
1940:L P[9998] 250mm/sec FINE;
1941:L P[9999] 250mm/sec CNT100;
1942:L P[10000] 250mm/sec CNT100;
1943:L P[10001] 250mm/sec FINE;
1944:L P[10002] 250mm/sec CNT100;
1945:L P[10003] 250mm/sec CNT100;
1946:L P[10004] 250mm/sec FINE;
1947:L P[10005] 250mm/sec CNT100;
1948:L P[10006] 250mm/sec CNT100;
1949:L P[10007] 250mm/sec FINE;
1950:L P[10008] 250mm/sec CNT100;
1951:L P[10009] 250mm/sec CNT100;
1952:L P[10010] 250mm/sec FINE;
1953:L P[10011] 250mm/sec CNT100;
1954:L P[10012] 250mm/sec CNT100;
1955:L P[10013] 250mm/sec FINE;
1956:L P[10014] 250mm/sec CNT100;
1957:L P[10015] 250mm/sec CNT100;
1958:L P[10016] 250mm/sec FINE;
1959:L P[10017] 250mm/sec CNT100;
1960:L P[10018] 250mm/sec CNT100;
1961:L P[10019] 250mm/sec FINE;
1962:L P[10020] 250mm/sec CNT100;
1963:L P[10021] 250mm/sec CNT100;
1964:L P[10022] 250mm/sec FINE;
1965:L P[10023] 250mm/sec CNT100;
1966:L P[10024] 250mm/sec CNT100;
1967:L P[10025] 250mm/sec FINE;
1968:L P[10026] 250mm/sec CNT100;
1969:L P[10027] 250mm/sec CNT100;
1970:L P[10028] 250mm/sec FINE;
1971:L P[10029] 250mm/sec CNT100;
1972:L P[10030] 250mm/sec CNT100;
1973:L P[10031] 250mm/sec FINE;
1974:L P[10032] 250mm/sec CNT100;
1975:L P[10033] 250mm/sec CNT100;
1976:L P[10034] 250mm/sec FINE;
1977:L P[10035] 250mm/sec CNT100;
1978:L P[10036] 250mm/sec CNT100;
1979:L P[10037] 250mm/sec FINE;
1980:L P[10038] 250mm/sec CNT100;
1981:L P[10039] 250mm/sec CNT100;
1982:L P[10040] 250mm/sec FINE;
1983:L P[10041] 250mm/sec CNT100;
1984:L P[10042] 250mm/sec CNT100;
1985:L P[10043] 250mm/sec FINE;
1986:L P[10044] 250mm/sec CNT100;
1987:L P[10045] 250mm/sec CNT100;
1988:L P[10046] 250mm/sec FINE;
1989:L P[10047] 250mm/sec CNT100;
1990:L P[10048] 250mm/sec CNT100;
1991:L P[10049] 250mm/sec FINE;
1992:L P[10050] 250mm/sec CNT100;
1993:L P[10051] 250mm/sec CNT100;
1994:L P[10052] 250mm/sec FINE;
1995:L P[10053] 250mm/sec CNT100;
1996:L P[10054] 250mm/sec CNT100;
1997:L P[10055] 250mm/sec FINE;
1998:L P[10056] 250mm/sec CNT100;
1999:L P[10057] 250mm/sec CNT100;
2000:L P[10058] 250mm/sec FINE;
2001:L P[10059] 250mm/sec CNT100;
2002:L P[10060] 250mm/sec CNT100;
2003:L P[10061] 250mm/sec FINE;
2004:L P[10062] 250mm/sec CNT100;
2005:L P[10063] 250mm/sec CNT100;
2006:L P[10064] 250mm/sec FINE;
2007:L P[10065] 250mm/sec CNT100;
2008:L P[10066] 250mm/sec CNT100;
2009:L P[10067] 250mm/sec FINE;
2010:L P[10068] 250mm/sec CNT100;
2011:L P[10069] 250mm/sec CNT100;
2012:L P[10070] 250mm/sec FINE;
2013:L P[10071] 250mm/sec CNT100;
2014:L P[10072] 250mm/sec CNT100;
2015:L P[10073] 250mm/sec FINE;
2016:L P[10074] 250mm/sec CNT100;
2017:L P[10075] 250mm/sec CNT100;
2018:L P[10076] 250mm/sec FINE;
2019:L P[10077] 250mm/sec CNT100;
2020:L P[10078] 250mm/sec CNT100;
2021:L P[10079] 250mm/sec FINE;
2022:L P[10080] 250mm/sec CNT100;
2023:L P[10081] 250mm/sec CNT100;
2024:L P[10082] 250mm/sec FINE;
2025:L P[10083] 250mm/sec CNT100;
2026:L P[10084] 250mm/sec CNT100;
2027:L P[10085] 250mm/sec FINE;
2028:L P[10086] 250mm/sec CNT100;
2029:L P[10087] 250mm/sec CNT100;
2030:L P[10088] 250mm/sec FINE;
2031:L P[10089] 250mm/sec CNT100;
2032:L P[10090] 250mm/sec CNT100;
2033:L P[10091] 250mm/sec FINE;
2034:L P[10092] 250mm/sec CNT100;
2035:L P[10093] 250mm/sec CNT100;
2036:L P[10094] 250mm/sec FINE;
2037:L P[10095] 250mm/sec CNT100;
2038:L P[10096] 250mm/sec CNT100;
2039:L P[10097] 250mm/sec FINE;
2040:L P[10098] 250mm/sec CNT100;
2041:L P[10099] 250mm/sec CNT100;
2042:L P[10100] 250mm/sec FINE;
2043:L P[10101] 250mm/sec CNT100;
2044:L P[10102] 250mm/sec CNT100;
2045:L P[10103] 250mm/sec FINE;
2046:L P[10104] 250mm/sec CNT100;
2047:L P[10105] 250mm/sec CNT100;
2048:L P[10106] 250mm/sec FINE;
2049:L P[10107] 250mm/sec CNT100;
2050:L P[10108] 250mm/sec CNT100;
2051:L P[10109] 250mm/sec FINE;
2052:L P[10110] 250mm/sec CNT100;
2053:L P[10111] 250mm/sec CNT100;
2054:L P[10112] 250mm/sec FINE;
2055:L P[10113] 250mm/sec CNT100;
2056:L P[10114] 250mm/sec CNT100;
2057:L P[10115] 250mm/sec FINE;
2058:L P[10116] 250mm/sec CNT100;
2059:L P[10117] 250mm/sec CNT100;
2060:L P[10118] 250mm/sec FINE;
2061:L P[10119] 250mm/sec CNT100;
2062:L P[10120] 250mm/sec CNT100;
2063:L P[10121] 250mm/sec FINE;
2064:L P[10122] 250mm/sec CNT100;
2065:L P[10123] 250mm/sec CNT100;
2066:L P[10124] 250mm/sec FINE;
2067:L P[10125] 250mm/sec CNT100;
2068:L P[10126] 250mm/sec CNT100;
2069:L P[10127] 250mm/sec FINE;
2070:L P[10128] 250mm/sec CNT100;
2071:L P[10129] 250mm/sec CNT100;
2072:L P[10130] 250mm/sec FINE;
2073:L P[10131] 250mm/sec CNT100;
2074:L P[10132] 250mm/sec CNT100;
2075:L P[10133] 250mm/sec FINE;
2076:L P[10134] 250mm/sec CNT100;
2077:L P[10135] 250mm/sec CNT100;
2078:L P[10136] 250mm/sec FINE;
2079:L P[10137] 250mm/sec CNT100;
2080:L P[10138] 250mm/sec CNT100;
2081:L P[10139] 250mm/sec FINE;
2082:L P[10140] 250mm/sec CNT100;
2083:L P[10141] 250mm/sec CNT100;
2084:L P[10142] 250mm/sec FINE;
2085:L P[10143] 250mm/sec CNT100;
2086:L P[10144] 250mm/sec CNT100;
2087:L P[10145] 250mm/sec FINE;
2088:L P[10146] 250mm/sec CNT100;
2089:L P[10147] 250mm/sec CNT100;
2090:L P[10148] 250mm/sec FINE;
2091:L P[10149] 250mm/sec CNT100;
2092:L P[10150] 250mm/sec CNT100;
2093:L P[10151] 250mm/sec FINE;
2094:L P[10152] 250mm/sec CNT100;
2095:L P[10153] 250mm/sec CNT100;
2096:L P[10154] 250mm/sec FINE;
2097:L P[10155] 250mm/sec CNT100;
2098:L P[10156] 250mm/sec CNT100;
2099:L P[10157] 250mm/sec FINE;
2100:L P[10158] 250mm/sec CNT100;
2101:L P[10159] 250mm/sec CNT100;
2102:L P[10160] 250mm/sec FINE;
2103:L P[10161] 250mm/sec CNT100;
2104:L P[10162] 250mm/sec CNT100;
2105:L P[10163] 250mm/sec FINE;
2106:L P[10164] 250mm/sec CNT100;
2107:L P[10165] 250mm/sec CNT100;
2108:L P[10166] 250mm/sec FINE;
2109:L P[10167] 250mm/sec CNT100;
2110:L P[10168] 250mm/sec CNT100;
2111:L P[10169] 250mm/sec FINE;
2112:L P[10170] 250mm/sec CNT100;
2113:L P[10171] 250mm/sec CNT100;
2114:L P[10172] 250mm/sec FINE;
2115:L P[10173] 250mm/sec CNT100;
2116:L P[10174] 250mm/sec CNT100;
2117:L P[10175] 250mm/sec FINE;
2118:L P[10176] 250mm/sec CNT100;
2119:L P[10177] 250mm/sec CNT100;
2120:L P[10178] 250mm/sec FINE;
2121:L P[10179] 250mm/sec CNT100;
2122:L P[10180] 250mm/sec CNT100;
2123:L P[10181] 250mm/sec FINE;
2124:L P[10182] 250mm/sec CNT100;
2125:L P[10183] 250mm/sec CNT100;
2126:L P[10184] 250mm/sec FINE;
2127:L P[10185] 250mm/sec CNT100;
2128:L P[10186] 250mm/sec CNT100;
2129:L P[10187] 250mm/sec FINE;
2130:L P[10188] 250mm/sec CNT100;
2131:L P[10189] 250mm/sec CNT100;
2132:L P[10190] 250mm/sec FINE;
2133:L P[10191] 250mm/sec CNT100;
2134:L P[10192] 250mm/sec CNT100;
2135:L P[10193] 250mm/sec FINE;
2136:L P[10194] 250mm/sec CNT100;
2137:L P[10195] 250mm/sec CNT100;
2138:L P[10196] 250mm/sec FINE;
2139:L P[10197] 250mm/sec CNT100;
2140:L P[10198] 250mm/sec CNT100;
2141:L P[10199] 250mm/sec FINE;
2142:L P[10200] 250mm/sec CNT100;
2143:L P[10201] 250mm/sec CNT100;
2144:L P[10202] 250mm/sec FINE;
2145:L P[10203] 250mm/sec CNT100;
2146:L P[10204] 250mm/sec CNT100;
2147:L P[10205] 250mm/sec FINE;
2148:L P[10206] 250mm/sec CNT100;
2149:L P[10207] 250mm/sec CNT100;
2150:L P[10208] 250mm/sec FINE;
2151:L P[10209] 250mm/sec CNT100;
2152:L P[10210] 250mm/sec CNT100;
2153:L P[10211] 250mm/sec FINE;
2154:L P[10212] 250mm/sec CNT100;
2155:L P[10213] 250mm/sec CNT100;
2156:L P[10214] 250mm/sec FINE;
2157:L P[10215] 250mm/sec CNT100;
2158:L P[10216] 250mm/sec CNT100;
2159:L P[10217] 250mm/sec FINE;
2160:L P[10218] 250mm/sec CNT100;
2161:L P[10219] 250mm/sec CNT100;
2162:L P[10220] 250mm/sec FINE;
2163:L P[10221] 250mm/sec CNT100;
2164:L P[10222] 250mm/sec CNT100;
2165:L P[10223] 250mm/sec FINE;
2166:L P[10224] 250mm/sec CNT100;
2167:L P[10225] 250mm/sec CNT100;
2168:L P[10226] 250mm/sec FINE;
2169:L P[10227] 250mm/sec CNT100;
2170:L P[10228] 250mm/sec CNT100;
2171:L P[10229] 250mm/sec FINE;
2172:L P[10230] 250mm/sec CNT100;
2173:L P[10231] 250mm/sec CNT100;
2174:L P[10232] 250mm/sec FINE;
2175:L P[10233] 250mm/sec CNT100;
2176:L P[10234] 250mm/sec CNT100;
2177:L P[10235] 250mm/sec FINE;
2178:L P[10236] 250mm/sec CNT100;
2179:L P[10237] 250mm/sec CNT100;
2180:L P[10238] 250mm/sec FINE;
2181:L P[10239] 250mm/sec CNT100;
2182:L P[10240] 250mm/sec CNT100;
2183:L P[10241] 250mm/sec FINE;
2184:L P[10242] 250mm/sec CNT100;
2185:L P[10243] 250mm/sec CNT100;
2186:L P[10244] 250mm/sec FINE;
2187:L P[10245] 250mm/sec CNT100;
2188:L P[10246] 250mm/sec CNT100;
2189:L P[10247] 250mm/sec FINE;
2190:L P[10248] 250mm/sec CNT100;
2191:L P[10249] 250mm/sec CNT100;
2192:L P[10250] 250mm/sec FINE;
2193:L P[10251] 250mm/sec CNT100;
2194:L P[10252] 250mm/sec CNT100;
2195:L P[10253] 250mm/sec FINE;
2196:L P[10254] 250mm/sec CNT100;
2197:L P[10255] 250mm/sec CNT100;
2198:L P[10256] 250mm/sec FINE;
2199:L P[10257] 250mm/sec CNT100;
2200:L P[10258] 250mm/sec CNT100;
2201:L P[10259] 250mm/sec FINE;
2202:L P[10260] 250mm/sec CNT100;
2203:L P[10261] 250mm/sec CNT100;
2204:L P[10262] 250mm/sec FINE;
2205:L P[10263] 250mm/sec CNT100;
2206:L P[10264] 250mm/sec CNT100;
2207:L P[10265] 250mm/sec FINE;
2208:L P[10266] 250mm/sec CNT100;
2209:L P[10267] 250mm/sec CNT100;
2210:L P[10268] 250mm/sec FINE;
2211:L P[10269] 250mm/sec CNT100;
2212:L P[10270] 250mm/sec CNT100;
2213:L P[10271] 250mm/sec FINE;
2214:L P[10272] 250mm/sec CNT100;
2215:L P[10273] 250mm/sec CNT100;
2216:L P[10274] 250mm/sec FINE;
2217:L P[10275] 250mm/sec CNT100;
2218:L P[10276] 250mm/sec CNT100;
2219:L P[10277] 250mm/sec FINE;
2220:L P[10278] 250mm/sec CNT100;
2221:L P[10279] 250mm/sec CNT100;
2222:L P[10280] 250mm/sec FINE;
2223:L P[10281] 250mm/sec CNT100;
2224:L P[10282] 250mm/sec CNT100;
2225:L P[10283] 250mm/sec FINE;
2226:L P[10284] 250mm/sec CNT100;
2227:L P[10285] 250mm/sec CNT100;
2228:L P[10286] 250mm/sec FINE;
2229:L P[10287] 250mm/sec CNT100;
2230:L P[10288] 250mm/sec CNT100;
2231:L P[10289] 250mm/sec FINE;
2232:L P[10290] 250mm/sec CNT100;
2233:L P[10291] 250mm/sec CNT100;
2234:L P[10292] 250mm/sec FINE;
2235:L P[10293] 250mm/sec CNT100;
2236:L P[10294] 250mm/sec CNT100;
2237:L P[10295] 250mm/sec FINE;
2238:L P[10296] 250mm/sec CNT100;
2239:L P[10297] 250mm/sec CNT100;
2240:L P[10298] 250mm/sec FINE;
2241:L P[10299] 250mm/sec CNT100;
2242:L P[10300] 250mm/sec CNT100;
2243:L P[10301] 250mm/sec FINE;
2244:L P[10302] 250mm/sec CNT100;
2245:L P[10303] 250mm/sec CNT100;
2246:L P[10304] 250mm/sec FINE;
2247:L P[10305] 250mm/sec CNT100;
2248:L P[10306] 250mm/sec CNT100;
2249:L P[10307] 250mm/sec FINE;
2250:L P[10308] 250mm/sec CNT100;
2251:L P[10309] 250mm/sec CNT100;
2252:L P[10310] 250mm/sec FINE;
2253:L P[10311] 250mm/sec CNT100;
2254:L P[10312] 250mm/sec CNT100;
2255:L P[10313] 250mm/sec FINE;
2256:L P[10314] 250mm/sec CNT100;
2257:L P[10315] 250mm/sec CNT100;
2258:L P[10316] 250mm/sec FINE;
2259:L P[10317] 250mm/sec CNT100;
2260:L P[10318] 250mm/sec CNT100;
2261:L P[10319] 250mm/sec FINE;
2262:L P[10320] 250mm/sec CNT100;
2263:L P[10321] 250mm/sec CNT100;
2264:L P[10322] 250mm/sec FINE;
2265:L P[10323] 250mm/sec CNT100;
2266:L P[10324] 250mm/sec CNT100;
2267:L P[10325] 250mm/sec FINE;
2268:L P[10326] 250mm/sec CNT100;
2269:L P[10327] 250mm/sec CNT100;
2270:L P[10328] 250mm/sec FINE;
2271:L P[10329] 250mm/sec CNT100;
2272:L P[10330] 250mm/sec CNT100;
2273:L P[10331] 250mm/sec FINE;
2274:L P[10332] 250mm/sec CNT100;
2275:L P[10333] 250mm/sec CNT100;
2276:L P[10334] 250mm/sec FINE;
2277:L P[10335] 250mm/sec CNT100;
2278:L P[10336] 250mm/sec CNT100;
2279:L P[10337] 250mm/sec FINE;
2280:L P[10338] 250mm/sec CNT100;
2281:L P[10339] 250mm/sec CNT100;
2282:L P[10340] 250mm/sec FINE;
2283:L P[10341] 250mm/sec CNT100;
2284:L P[10342] 250mm/sec CNT100;
2285:L P[10343] 250mm/sec FINE;
2286:L P[10344] 250mm/sec CNT100;
2287:L P[10345] 250mm/sec CNT100;
2288:L P[10346] 250mm/sec FINE;
2289:L P[10347] 250mm/sec CNT100;
2290:L P[10348] 250mm/sec CNT100;
2291:L P[10349] 250mm/sec FINE;
2292:L P[10350] 250mm/sec CNT100;
2293:L P[10351] 250mm/sec CNT100;
2294:L P[10352] 250mm/sec FINE;
2295:L P[10353] 250mm/sec CNT100;
2296:L P[10354] 250mm/sec CNT100;
2297:L P[10355] 250mm/sec FINE;
2298:L P[10356] 250mm/sec CNT100;
2299:L P[10357] 250mm/sec CNT100;
2300:L P[10358] 250mm/sec FINE;
2301:L P[10359] 250mm/sec CNT100;
2302:L P[10360] 250mm/sec CNT100;
2303:L P[10361] 250mm/sec FINE;
2304:L P[10362] 250mm/sec CNT100;
2305:L P[10363] 250mm/sec CNT100;
2306:L P[10364] 250mm/sec FINE;
2307:L P[10365] 250mm/sec CNT100;
2308:L P[10366] 250mm/sec CNT100;
2309:L P[10367] 250mm/sec FINE;
2310:L P[10368] 250mm/sec CNT100;
2311:L P[10369] 250mm/sec CNT100;
2312:L P[10370] 250mm/sec FINE;
2313:L P[10371] 250mm/sec CNT100;
2314:L P[10372] 250mm/sec CNT100;
2315:L P[10373] 250mm/sec FINE;
2316:L P[10374] 250mm/sec CNT100;
2317:L P[10375] 250mm/sec CNT100;
2318:L P[10376] 250mm/sec FINE;
2319:L P[10377] 250mm/sec CNT100;
2320:L P[10378] 250mm/sec CNT100;
2321:L P[10379] 250mm/sec FINE;
2322:L P[10380] 250mm/sec CNT100;
2323:L P[10381] 250mm/sec CNT100;
2324:L P[10382] 250mm/sec FINE;
2325:L P[10383] 250mm/sec CNT100;
2326:L P[10384] 250mm/sec CNT100;
2327:L P[10385] 250mm/sec FINE;
2328:L P[10386] 250mm/sec CNT100;
2329:L P[10387] 250mm/sec CNT100;
2330:L P[10388] 250mm/sec FINE;
2331:L P[10389] 250mm/sec CNT100;
2332:L P[10390] 250mm/sec CNT100;
2333:L P[10391] 250mm/sec FINE;
2334:L P[10392] 250mm/sec CNT100;
2335:L P[10393] 250mm/sec CNT100;
2336:L P[10394] 250mm/sec FINE;
2337:L P[10395] 250mm/sec CNT100;
2338:L P[10396] 250mm/sec CNT100;
2339:L P[10397] 250mm/sec FINE;
2340:L P[10398] 250mm/sec CNT100;
2341:L P[10399] 250mm/sec CNT100;
2342:L P[10400] 250mm/sec FINE;
2343:L P[10401] 250mm/sec CNT100;
2344:L P[10402] 250mm/sec CNT100;
2345:L P[10403] 250mm/sec FINE;
2346:L P[10404] 250mm/sec CNT100;
2347:L P[10405] 250mm/sec CNT100;
2348:L P[10406] 250mm/sec FINE;
2349:L P[10407] 250mm/sec CNT100;
2350:L P[10408] 250mm/sec CNT100;
2351:L P[10409] 250mm/sec FINE;
2352:L P[10410] 250mm/sec CNT100;
2353:L P[10411] 250mm/sec CNT100;
2354:L P[10412] 250mm/sec FINE;
2355:L P[10413] 250mm/sec CNT100;
2356:L P[10414] 250mm/sec CNT100;
2357:L P[10415] 250mm/sec FINE;
2358:L P[10416] 250mm/sec CNT100;
2359:L P[10417] 250mm/sec CNT100;
2360:L P[10418] 250mm/sec FINE;
2361:L P[10419] 250mm/sec CNT100;
2362:L P[10420] 250mm/sec CNT100;
2363:L P[10421] 250mm/sec FINE;
2364:L P[10422] 250mm/sec CNT100;
2365:L P[10423] 250mm/sec CNT100;
2366:L P[10424] 250mm/sec FINE;
2367:L P[10425] 250mm/sec CNT100;
2368:L P[10426] 250mm/sec CNT100;
2369:L P[10427] 250mm/sec FINE;
2370:L P[10428] 250mm/sec CNT100;
2371:L P[10429] 250mm/sec CNT100;
2372:L P[10430] 250mm/sec FINE;
2373:L P[10431] 250mm/sec CNT100;
2374:L P[10432] 250mm/sec CNT100;
2375:L P[10433] 250mm/sec FINE;
2376:L P[10434] 250mm/sec CNT100;
2377:L P[10435] 250mm/sec CNT100;
2378:L P[10436] 250mm/sec FINE;
2379:L P[10437] 250mm/sec CNT100;
2380:L P[10438] 250mm/sec CNT100;
2381:L P[10439] 250mm/sec FINE;
2382:L P[10440] 250mm/sec CNT100;
2383:L P[10441] 250mm/sec CNT100;
2384:L P[10442] 250mm/sec FINE;
2385:L P[10443] 250mm/sec CNT100;
2386:L P[10444] 250mm/sec CNT100;
2387:L P[10445] 250mm/sec FINE;
2388:L P[10446] 250mm/sec CNT100;
2389:L P[10447] 250mm/sec CNT100;
2390:L P[10448] 250mm/sec FINE;
2391:L P[10449] 250mm/sec CNT100;
2392:L P[10450] 250mm/sec CNT100;
2393:L P[10451] 250mm/sec FINE;
2394:L P[10452] 250mm/sec CNT100;
2395:L P[10453] 250mm/sec CNT100;
2396:L P[10454] 250mm/sec FINE;
2397:L P[10455] 250mm/sec CNT100;
2398:L P[10456] 250mm/sec CNT100;
2399:L P[10457] 250mm/sec FINE;
2400:L P[10458] 250mm/sec CNT100;
2401:L P[10459] 250mm/sec CNT100;
2402:L P[10460] 250mm/sec FINE;
2403:L P[10461] 250mm/sec CNT100;
2404:L P[10462] 250mm/sec CNT100;
2405:L P[10463] 250mm/sec FINE;
2406:L P[10464] 250mm/sec CNT100;
2407:L P[10465] 250mm/sec CNT100;
2408:L P[10466] 250mm/sec FINE;
2409:L P[10467] 250mm/sec CNT100;
2410:L P[10468] 250mm/sec CNT100;
2411:L P[10469] 250mm/sec FINE;
2412:L P[10470] 250mm/sec CNT100;
2413:L P[10471] 250mm/sec CNT100;
2414:L P[10472] 250mm/sec FINE;
2415:L P[10473] 250mm/sec CNT100;
2416:L P[10474] 250mm/sec CNT100;
2417:L P[10475] 250mm/sec FINE;
2418:L P[10476] 250mm/sec CNT100;
2419:L P[10477] 250mm/sec CNT100;
2420:L P[10478] 250mm/sec FINE;
2421:L P[10479] 250mm/sec CNT100;
2422:L P[10480] 250mm/sec CNT100;
2423:L P[10481] 250mm/sec FINE;
2424:L P[10482] 250mm/sec CNT100;
2425:L P[10483] 250mm/sec CNT100;
2426:L P[10484] 250mm/sec FINE;
2427:L P[10485] 250mm/sec CNT100;
2428:L P[10486] 250mm/sec CNT100;
2429:L P[10487] 250mm/sec FINE;
2430:L P[10488] 250mm/sec CNT100;
2431:L P[10489] 250mm/sec CNT100;
2432:L P[10490] 250mm/sec FINE;
2433:L P[10491] 250mm/sec CNT100;
2434:L P[10492] 250mm/sec CNT100;
2435:L P[10493] 250mm/sec FINE;
2436:L P[10494] 250mm/sec CNT100;
2437:L P[10495] 250mm/sec CNT100;
2438:L P[10496] 250mm/sec FINE;
2439:L P[10497] 250mm/sec CNT100;
2440:L P[10498] 250mm/sec CNT100;
2441:L P[10499] 250mm/sec FINE;
2442:L P[10500] 250mm/sec CNT100;
2443:L P[10501] 250mm/sec CNT100;
2444:L P[10502] 250mm/sec FINE;
2445:L P[10503] 250mm/sec CNT100;
2446:L P[10504] 250mm/sec CNT100;
2447:L P[10505] 250mm/sec FINE;
2448:L P[10506] 250mm/sec CNT100;
2449:L P[10507] 250mm/sec CNT100;
2450:L P[10508] 250mm/sec FINE;
2451:L P[10509] 250mm/sec CNT100;
2452:L P[10510] 250mm/sec CNT100;
2453:L P[10511] 250mm/sec FINE;
2454:L P[10512] 250mm/sec CNT100;
2455:L P[10513] 250mm/sec CNT100;
2456:L P[10514] 250mm/sec FINE;
2457:L P[10515] 250mm/sec CNT100;
2458:L P[10516] 250mm/sec CNT100;
2459:L P[10517] 250mm/sec FINE;
2460:L P[10518] 250mm/sec CNT100;
2461:L P[10519] 250mm/sec CNT100;
2462:L P[10520] 250mm/sec FINE;
2463:L P[10521] 250mm/sec CNT100;
2464:L P[10522] 250mm/sec CNT100;
2465:L P[10523] 250mm/sec FINE;
2466:L P[10524] 250mm/sec CNT100;
2467:L P[10525] 250mm/sec CNT100;
2468:L P[10526] 250mm/sec FINE;
2469:L P[10527] 250mm/sec CNT100;
2470:L P[10528] 250mm/sec CNT100;
2471:L P[10529] 250mm/sec FINE;
2472:L P[10530] 250mm/sec CNT100;
2473:L P[10531] 250mm/sec CNT100;
2474:L P[10532] 250mm/sec FINE;
2475:L P[10533] 250mm/sec CNT100;
2476:L P[10534] 250mm/sec CNT100;
2477:L P[10535] 250mm/sec FINE;
2478:L P[10536] 250mm/sec CNT100;
2479:L P[10537] 250mm/sec CNT100;
2480:L P[10538] 250mm/sec FINE;
2481:L P[10539] 250mm/sec CNT100;
2482:L P[10540] 250mm/sec CNT100;
2483:L P[10541] 250mm/sec FINE;
2484:L P[10542] 250mm/sec CNT100;
2485:L P[10543] 250mm/sec CNT100;
2486:L P[10544] 250mm/sec FINE;
2487:L P[10545] 250mm/sec CNT100;
2488:L P[10546] 250mm/sec CNT100;
2489:L P[10547] 250mm/sec FINE;
2490:L P[10548] 250mm/sec CNT100;
2491:L P[10549] 250mm/sec CNT100;
2492:L P[10550] 250mm/sec FINE;
2493:L P[10551] 250mm/sec CNT100;
2494:L P[10552] 250mm/sec CNT100;
2495:L P[10553] 250mm/sec FINE;
2496:L P[10554] 250mm/sec CNT100;
2497:L P[10555] 250mm/sec CNT100;
2498:L P[10556] 250mm/sec FINE;
2499:L P[10557] 250mm/sec CNT100;
2500:L P[10558] 250mm/sec CNT100;
2501:L P[10559] 250mm/sec FINE;
2502:L P[10560] 250mm/sec CNT100;
2503:L P[10561] 250mm/sec CNT100;
2504:L P[10562] 250mm/sec FINE;
2505:L P[10563] 250mm/sec CNT100;
2506:L P[10564] 250mm/sec CNT100;
2507:L P[10565] 250mm/sec FINE;
2508:L P[10566] 250mm/sec CNT100;
2509:L P[10567] 250mm/sec CNT100;
2510:L P[10568] 250mm/sec FINE;
2511:L P[10569] 250mm/sec CNT100;
2512:L P[10570] 250mm/sec CNT100;
2513:L P[10571] 250mm/sec FINE;
2514:L P[10572] 250mm/sec CNT100;
2515:L P[10573] 250mm/sec CNT100;
2516:L P[10574] 250mm/sec FINE;
2517:L P[10575] 250mm/sec CNT100;
2518:L P[10576] 250mm/sec CNT100;
2519:L P[10577] 250mm/sec FINE;
2520:L P[10578] 250mm/sec CNT100;
2521:L P[10579] 250mm/sec CNT100;
2522:L P[10580] 250mm/sec FINE;
2523:L P[10581] 250mm/sec CNT100;
2524:L P[10582] 250mm/sec CNT100;
2525:L P[10583] 250mm/sec FINE;
2526:L P[10584] 250mm/sec CNT100;
2527:L P[10585] 250mm/sec CNT100;
2528:L P[10586] 250mm/sec FINE;
2529:L P[10587] 250mm/sec CNT100;
2530:L P[10588] 250mm/sec CNT100;
2531:L P[10589] 250mm/sec FINE;
2532:L P[10590] 250mm/sec CNT100;
2533:L P[10591] 250mm/sec CNT100;
2534:L P[10592] 250mm/sec FINE;
2535:L P[10593] 250mm/sec CNT100;
2536:L P[10594] 250mm/sec CNT100;
2537:L P[10595] 250mm/sec FINE;
2538:L P[10596] 250mm/sec CNT100;
2539:L P[10597] 250mm/sec CNT100;
2540:L P[10598] 250mm/sec FINE;
2541:L P[10599] 250mm/sec CNT100;
2542:L P[10600] 250mm/sec CNT100;
2543:L P[10601] 250mm/sec FINE;
2544:L P[10602] 250mm/sec CNT100;
2545:L P[10603] 250mm/sec CNT100;
2546:L P[10604] 250mm/sec FINE;
2547:L P[10605] 250mm/sec CNT100;
2548:L P[10606] 250mm/sec CNT100;
2549:L P[10607] 250mm/sec FINE;
2550:L P[10608] 250mm/sec CNT100;
2551:L P[10609] 250mm/sec CNT100;
2552:L P[10610] 250mm/sec FINE;
2553:L P[10611] 250mm/sec CNT100;
2554:L P[10612] 250mm/sec CNT100;
2555:L P[10613] 250mm/sec FINE;
2556:L P[10614] 250mm/sec CNT100;
2557:L P[10615] 250mm/sec CNT100;
2558:L P[10616] 250mm/sec FINE;
2559:L P[10617] 250mm/sec CNT100;
2560:L P[10618] 250mm/sec CNT100;
2561:L P[10619] 250mm/sec FINE;
2562:L P[10620] 250mm/sec CNT100;
2563:L P[10621] 250mm/sec CNT100;
2564:L P[10622] 250mm/sec FINE;
2565:L P[10623] 250mm/sec CNT100;
2566:L P[10624] 250mm/sec CNT100;
2567:L P[10625] 250mm/sec FINE;
2568:L P[10626] 250mm/sec CNT100;
2569:L P[10627] 250mm/sec CNT100;
2570:L P[10628] 250mm/sec FINE;
2571:L P[10629] 250mm/sec CNT100;
2572:L P[10630] 250mm/sec CNT100;
2573:L P[10631] 250mm/sec FINE;
2574:L P[10632] 250mm/sec CNT100;
2575:L P[10633] 250mm/sec CNT100;
2576:L P[10634] 250mm/sec FINE;
2577:L P[10635] 250mm/sec CNT100;
2578:L P[10636] 250mm/sec CNT100;
2579:L P[10637] 250mm/sec FINE;
2580:L P[10638] 250mm/sec CNT100;
2581:L P[10639] 250mm/sec CNT100;
2582:L P[10640] 250mm/sec FINE;
2583:L P[10641] 250mm/sec CNT100;
2584:L P[10642] 250mm/sec CNT100;
2585:L P[10643] 250mm/sec FINE;
2586:L P[10644] 250mm/sec CNT100;
2587:L P[10645] 250mm/sec CNT100;
2588:L P[10646] 250mm/sec FINE;
2589:L P[10647] 250mm/sec CNT100;
2590:L P[10648] 250mm/sec CNT100;
2591:L P[10649] 250mm/sec FINE;
2592:L P[10650] 250mm/sec CNT100;
2593:L P[10651] 250mm/sec CNT100;
2594:L P[10652] 250mm/sec FINE;
2595:L P[10653] 250mm/sec CNT100;
2596:L P[10654] 250mm/sec CNT100;
2597:L P[10655] 250mm/sec FINE;
2598:L P[10656] 250mm/sec CNT100;
2599:L P[10657] 250mm/sec CNT100;
2600:L P[10658] 250mm/sec FINE;
2601:L P[10659] 250mm/sec CNT100;
2602:L P[10660] 250mm/sec CNT100;
2603:L P[10661] 250mm/sec FINE;
2604:L P[10662] 250mm/sec CNT100;
2605:L P[10663] 250mm/sec CNT100;
2606:L P[10664] 250mm/sec FINE;
2607:L P[10665] 250mm/sec CNT100;
2608:L P[10666] 250mm/sec CNT100;
2609:L P[10667] 250mm/sec FINE;
2610:L P[10668] 250mm/sec CNT100;
2611:L P[10669] 250mm/sec CNT100;
2612:L P[10670] 250mm/sec FINE;
2613:L P[10671] 250mm/sec CNT100;
2614:L P[10672] 250mm/sec CNT100;
2615:L P[10673] 250mm/sec FINE;
2616:L P[10674] 250mm/sec CNT100;
2617:L P[10675] 250mm/sec CNT100;
2618:L P[10676] 250mm/sec FINE;
2619:L P[10677] 250mm/sec CNT100;
2620:L P[10678] 250mm/sec CNT100;
2621:L P[10679] 250mm/sec FINE;
2622:L P[10680] 250mm/sec CNT100;
2623:L P[10681] 250mm/sec CNT100;
2624:L P[10682] 250mm/sec FINE;
2625:L P[10683] 250mm/sec CNT100;
2626:L P[10684] 250mm/sec CNT100;
2627:L P[10685] 250mm/sec FINE;
2628:L P[10686] 250mm/sec CNT100;
2629:L P[10687] 250mm/sec CNT100;
2630:L P[10688] 250mm/sec FINE;
2631:L P[10689] 250mm/sec CNT100;
2632:L P[10690] 250mm/sec CNT100;
2633:L P[10691] 250mm/sec FINE;
2634:L P[10692] 250mm/sec CNT100;
2635:L P[10693] 250mm/sec CNT100;
2636:L P[10694] 250mm/sec FINE;
2637:L P[10695] 250mm/sec CNT100;
2638:L P[10696] 250mm/sec CNT100;
2639:L P[10697] 250mm/sec FINE;
2640:L P[10698] 250mm/sec CNT100;
2641:L P[10699] 250mm/sec CNT100;
2642:L P[10700] 250mm/sec FINE;
2643:L P[10701] 250mm/sec CNT100;
2644:L P[10702] 250mm/sec CNT100;
2645:L P[10703] 250mm/sec FINE;
2646:L P[10704] 250mm/sec CNT100;
2647:L P[10705] 250mm/sec CNT100;
2648:L P[10706] 250mm/sec FINE;
2649:L P[10707] 250mm/sec CNT100;
2650:L P[10708] 250mm/sec CNT100;
2651:L P[10709] 250mm/sec FINE;
2652:L P[10710] 250mm/sec CNT100;
2653:L P[10711] 250mm/sec CNT100;
2654:L P[10712] 250mm/sec FINE;
2655:L P[10713] 250mm/sec CNT100;
2656:L P[10714] 250mm/sec CNT100;
2657:L P[10715] 250mm/sec FINE;
2658:L P[10716] 250mm/sec CNT100;
2659:L P[10717] 250mm/sec CNT100;
2660:L P[10718] 250mm/sec FINE;
2661:L P[10719] 250mm/sec CNT100;
2662:L P[10720] 250mm/sec CNT100;
2663:L P[10721] 250mm/sec FINE;
2664:L P[10722] 250mm/sec CNT100;
2665:L P[10723] 250mm/sec CNT100;
2666:L P[10724] 250mm/sec FINE;
2667:L P[10725] 250mm/sec CNT100;
2668:L P[10726] 250mm/sec CNT100;
2669:L P[10727] 250mm/sec FINE;
2670:L P[10728] 250mm/sec CNT100;
2671:L P[10729] 250mm/sec CNT100;
2672:L P[10730] 250mm/sec FINE;
2673:L P[10731] 250mm/sec CNT100;
2674:L P[10732] 250mm/sec CNT100;
2675:L P[10733] 250mm/sec FINE;
2676:L P[10734] 250mm/sec CNT100;
2677:L P[10735] 250mm/sec CNT100;
2678:L P[10736] 250mm/sec FINE;
2679:L P[10737] 250mm/sec CNT100;
2680:L P[10738] 250mm/sec CNT100;
2681:L P[10739] 250mm/sec FINE;
2682:L P[10740] 250mm/sec CNT100;
2683:L P[10741] 250mm/sec CNT100;
2684:L P[10742] 250mm/sec FINE;
2685:L P[10743] 250mm/sec CNT100;
2686:L P[10744] 250mm/sec CNT100;
2687:L P[10745] 250mm/sec FINE;
2688:L P[10746] 250mm/sec CNT100;
2689:L P[10747] 250mm/sec CNT100;
2690:L P[10748] 250mm/sec FINE;
2691:L P[10749] 250mm/sec CNT100;
2692:L P[10750] 250mm/sec CNT100;
2693:L P[10751] 250mm/sec FINE;
2694:L P[10752] 250mm/sec CNT100;
2695:L P[10753] 250mm/sec CNT100;
2696:L P[10754] 250mm/sec FINE;
2697:L P[10755] 250mm/sec CNT100;
2698:L P[10756] 250mm/sec CNT100;
2699:L P[10757] 250mm/sec FINE;
2700:L P[10758] 250mm/sec CNT100;
2701:L P[10759] 250mm/sec CNT100;
2702:L P[10760] 250mm/sec FINE;
2703:L P[10761] 250mm/sec CNT100;
2704:L P[10762] 250mm/sec CNT100;
2705:L P[10763] 250mm/sec FINE;
2706:L P[10764] 250mm/sec CNT100;
2707:L P[10765] 250mm/sec CNT100;
2708:L P[10766] 250mm/sec FINE;
2709:L P[10767] 250mm/sec CNT100;
2710:L P[10768] 250mm/sec CNT100;
2711:L P[10769] 250mm/sec FINE;
2712:L P[10770] 250mm/sec CNT100;
2713:L P[10771] 250mm/sec CNT100;
2714:L P[10772] 250mm/sec FINE;
2715:L P[10773] 250mm/sec CNT100;
2716:L P[10774] 250mm/sec CNT100;
2717:L P[10775] 250mm/sec FINE;
2718:L P[10776] 250mm/sec CNT100;
2719:L P[10777] 250mm/sec CNT100;
2720:L P[10778] 250mm/sec FINE;
2721:L P[10779] 250mm/sec CNT100;
2722:L P[10780] 250mm/sec CNT100;
2723:L P[10781] 250mm/sec FINE;
2724:L P[10782] 250mm/sec CNT100;
2725:L P[10783] 250mm/sec CNT100;
2726:L P[10784] 250mm/sec FINE;
2727:L P[10785] 250mm/sec CNT100;
2728:L P[10786] 250mm/sec CNT100;
2729:L P[10787] 250mm/sec FINE;
2730:L P[10788] 250mm/sec CNT100;
2731:L P[10789] 250mm/sec CNT100;
2732:L P[10790] 250mm/sec FINE;
2733:L P[10791] 250mm/sec CNT100;
2734:L P[10792] 250mm/sec CNT100;
2735:L P[10793] 250mm/sec FINE;
2736:L P[10794] 250mm/sec CNT100;
2737:L P[10795] 250mm/sec CNT100;
2738:L P[10796] 250mm/sec FINE;
2739:L P[10797] 250mm/sec CNT100;
2740:L P[10798] 250mm/sec CNT100;
2741:L P[10799] 250mm/sec FINE;
2742:L P[10800] 250mm/sec CNT100;
2743:L P[10801] 250mm/sec CNT100;
2744:L P[10802] 250mm/sec FINE;
2745:L P[10803] 250mm/sec CNT100;
2746:L P[10804] 250mm/sec CNT100;
2747:L P[10805] 250mm/sec FINE;
2748:L P[10806] 250mm/sec CNT100;
2749:L P[10807] 250mm/sec CNT100;
2750:L P[10808] 250mm/sec FINE;
2751:L P[10809] 250mm/sec CNT100;
2752:L P[10810] 250mm/sec CNT100;
2753:L P[10811] 250mm/sec FINE;
2754:L P[10812] 250mm/sec CNT100;
2755:L P[10813] 250mm/sec CNT100;
2756:L P[10814] 250mm/sec FINE;
2757:L P[10815] 250mm/sec CNT100;
2758:L P[10816] 250mm/sec CNT100;
2759:L P[10817] 250mm/sec FINE;
2760:L P[10818] 250mm/sec CNT100;
2761:L P[10819] 250mm/sec CNT100;
2762:L P[10820] 250mm/sec FINE;
2763:L P[10821] 250mm/sec CNT100;
2764:L P[10822] 250mm/sec CNT100;
2765:L P[10823] 250mm/sec FINE;
2766:L P[10824] 250mm/sec CNT100;
2767:L P[10825] 250mm/sec CNT100;
2768:L P[10826] 250mm/sec FINE;
2769:L P[10827] 250mm/sec CNT100;
2770:L P[10828] 250mm/sec CNT100;
2771:L P[10829] 250mm/sec FINE;
2772:L P[10830] 250mm/sec CNT100;
2773:L P[10831] 250mm/sec CNT100;
2774:L P[10832] 250mm/sec FINE;
2775:L P[10833] 250mm/sec CNT100;
2776:L P[10834] 250mm/sec CNT100;
2777:L P[10835] 250mm/sec FINE;
2778:L P[10836] 250mm/sec CNT100;
2779:L P[10837] 250mm/sec CNT100;
2780:L P[10838] 250mm/sec FINE;
2781:L P[10839] 250mm/sec CNT100;
2782:L P[10840] 250mm/sec CNT100;
2783:L P[10841] 250mm/sec FINE;
2784:L P[10842] 250mm/sec CNT100;
2785:L P[10843] 250mm/sec CNT100;
2786:L P[10844] 250mm/sec FINE;
2787:L P[10845] 250mm/sec CNT100;
2788:L P[10846] 250mm/sec CNT100;
2789:L P[10847] 250mm/sec FINE;
2790:L P[10848] 250mm/sec CNT100;
2791:L P[10849] 250mm/sec CNT100;
2792:L P[10850] 250mm/sec FINE;
2793:L P[10851] 250mm/sec CNT100;
2794:L P[10852] 250mm/sec CNT100;
2795:L P[10853] 250mm/sec FINE;
2796:L P[10854] 250mm/sec CNT100;
2797:L P[10855] 250mm/sec CNT100;
2798:L P[10856] 250mm/sec FINE;
2799:L P[10857] 250mm/sec CNT100;
2800:L P[10858] 250mm/sec CNT100;
2801:L P[10859] 250mm/sec FINE;
2802:L P[10860] 250mm/sec CNT100;
2803:L P[10861] 250mm/sec CNT100;
2804:L P[10862] 250mm/sec FINE;
2805:L P[10863] 250mm/sec CNT100;
2806:L P[10864] 250mm/sec CNT100;
2807:L P[10865] 250mm/sec FINE;
2808:L P[10866] 250mm/sec CNT100;
2809:L P[10867] 250mm/sec CNT100;
2810:L P[10868] 250mm/sec FINE;
2811:L P[10869] 250mm/sec CNT100;
2812:L P[10870] 250mm/sec CNT100;
2813:L P[10871] 250mm/sec FINE;
2814:L P[10872] 250mm/sec CNT100;
2815:L P[10873] 250mm/sec CNT100;
2816:L P[10874] 250mm/sec FINE;
2817:L P[10875] 250mm/sec CNT100;
2818:L P[10876] 250mm/sec CNT100;
2819:L P[10877] 250mm/sec FINE;
2820:L P[10878] 250mm/sec CNT100;
2821:L P[10879] 250mm/sec CNT100;
2822:L P[10880] 250mm/sec FINE;
2823:L P[10881] 250mm/sec CNT100;
2824:L P[10882] 250mm/sec CNT100;
2825:L P[10883] 250mm/sec FINE;
2826:L P[10884] 250mm/sec CNT100;
2827:L P[10885] 250mm/sec CNT100;
2828:L P[10886] 250mm/sec FINE;
2829:L P[10887] 250mm/sec CNT100;
2830:L P[10888] 250mm/sec CNT100;
2831:L P[10889] 250mm/sec FINE;
2832:L P[10890] 250mm/sec CNT100;
2833:L P[10891] 250mm/sec CNT100;
2834:L P[10892] 250mm/sec FINE;
2835:L P[10893] 250mm/sec CNT100;
2836:L P[10894] 250mm/sec CNT100;
2837:L P[10895] 250mm/sec FINE;
2838:L P[10896] 250mm/sec CNT100;
2839:L P[10897] 250mm/sec CNT100;
2840:L P[10898] 250mm/sec FINE;
2841:L P[10899] 250mm/sec CNT100;
2842:L P[10900] 250mm/sec CNT100;
2843:L P[10901] 250mm/sec FINE;
2844:L P[10902] 250mm/sec CNT100;
2845:L P[10903] 250mm/sec CNT100;
2846:L P[10904] 250mm/sec FINE;
2847:L P[10905] 250mm/sec CNT100;
2848:L P[10906] 250mm/sec CNT100;
2849:L P[10907] 250mm/sec FINE;
2850:L P[10908] 250mm/sec CNT100;
2851:L P[10909] 250mm/sec CNT100;
2852:L P[10910] 250mm/sec FINE;
2853:L P[10911] 250mm/sec CNT100;
2854:L P[10912] 250mm/sec CNT100;
2855:L P[10913] 250mm/sec FINE;
2856:L P[10914] 250mm/sec CNT100;
2857:L P[10915] 250mm/sec CNT100;
2858:L P[10916] 250mm/sec FINE;
2859:L P[10917] 250mm/sec CNT100;
2860:L P[10918] 250mm/sec CNT100;
2861:L P[10919] 250mm/sec FINE;
2862:L P[10920] 250mm/sec CNT100;
2863:L P[10921] 250mm/sec CNT100;
2864:L P[10922] 250mm/sec FINE;
2865:L P[10923] 250mm/sec CNT100;
2866:L P[10924] 250mm/sec CNT100;
2867:L P[10925] 250mm/sec FINE;
2868:L P[10926] 250mm/sec CNT100;
2869:L P[10927] 250mm/sec CNT100;
2870:L P[10928] 250mm/sec FINE;
2871:L P[10929] 250mm/sec CNT100;
2872:L P[10930] 250mm/sec CNT100;
2873:L P[10931] 250mm/sec FINE;
2874:L P[10932] 250mm/sec CNT100;
2875:L P[10933] 250mm/sec CNT100;
2876:L P[10934] 250mm/sec FINE;
2877:L P[10935] 250mm/sec CNT100;
2878:L P[10936] 250mm/sec CNT100;
2879:L P[10937] 250mm/sec FINE;
2880:L P[10938] 250mm/sec CNT100;
2881:L P[10939] 250mm/sec CNT100;
2882:L P[10940] 250mm/sec FINE;
2883:L P[10941] 250mm/sec CNT100;
2884:L P[10942] 250mm/sec CNT100;
2885:L P[10943] 250mm/sec FINE;
2886:L P[10944] 250mm/sec CNT100;
2887:L P[10945] 250mm/sec CNT100;
2888:L P[10946] 250mm/sec FINE;
2889:L P[10947] 250mm/sec CNT100;
2890:L P[10948] 250mm/sec CNT100;
2891:L P[10949] 250mm/sec FINE;
2892:L P[10950] 250mm/sec CNT100;
2893:L P[10951] 250mm/sec CNT100;
2894:L P[10952] 250mm/sec FINE;
2895:L P[10953] 250mm/sec CNT100;
2896:L P[10954] 250mm/sec CNT100;
2897:L P[10955] 250mm/sec FINE;
2898:L P[10956] 250mm/sec CNT100;
2899:L P[10957] 250mm/sec CNT100;
2900:L P[10958] 250mm/sec FINE;
2901:L P[10959] 250mm/sec CNT100;
2902:L P[10960] 250mm/sec CNT100;
2903:L P[10961] 250mm/sec FINE;
2904:L P[10962] 250mm/sec CNT100;
2905:L P[10963] 250mm/sec CNT100;
2906:L P[10964] 250mm/sec FINE;
2907:L P[10965] 250mm/sec CNT100;
2908:L P[10966] 250mm/sec CNT100;
2909:L P[10967] 250mm/sec FINE;
2910:L P[10968] 250mm/sec CNT100;
2911:L P[10969] 250mm/sec CNT100;
2912:L P[10970] 250mm/sec FINE;
2913:L P[10971] 250mm/sec CNT100;
2914:L P[10972] 250mm/sec CNT100;
2915:L P[10973] 250mm/sec FINE;
2916:L P[10974] 250mm/sec CNT100;
2917:L P[10975] 250mm/sec CNT100;
2918:L P[10976] 250mm/sec FINE;
2919:L P[10977] 250mm/sec CNT100;
2920:L P[10978] 250mm/sec CNT100;
2921:L P[10979] 250mm/sec FINE;
2922:L P[10980] 250mm/sec CNT100;
2923:L P[10981] 250mm/sec CNT100;
2924:L P[10982] 250mm/sec FINE;
2925:L P[10983] 250mm/sec CNT100;
2926:L P[10984] 250mm/sec CNT100;
2927:L P[10985] 250mm/sec FINE;
2928:L P[10986] 250mm/sec CNT100;
2929:L P[10987] 250mm/sec CNT100;
2930:L P[10988] 250mm/sec FINE;
2931:L P[10989] 250mm/sec CNT100;
2932:L P[10990] 250mm/sec CNT100;
2933:L P[10991] 250mm/sec FINE;
2934:L P[10992] 250mm/sec CNT100;
2935:L P[10993] 250mm/sec CNT100;
2936:L P[10994] 250mm/sec FINE;
2937:L P[10995] 250mm/sec CNT100;
2938:L P[10996] 250mm/sec CNT100;
2939:L P[10997] 250mm/sec FINE;
2940:L P[10998] 250mm/sec CNT100;
2941:L P[10999] 250mm/sec CNT100;
2942:L P[11000] 250mm/sec FINE;
2943:L P[11001] 250mm/sec CNT100;
2944:L P[11002] 250mm/sec CNT100;
2945:L P[11003] 250mm/sec FINE;
2946:L P[11004] 250mm/sec CNT100;
2947:L P[11005] 250mm/sec CNT100;
2948:L P[11006] 250mm/sec FINE;
2949:L P[11007] 250mm/sec CNT100;
2950:L P[11008] 250mm/sec CNT100;
2951:L P[11009] 250mm/sec FINE;
2952:L P[11010] 250mm/sec CNT100;
2953:L P[11011] 250mm/sec CNT100;
2954:L P[11012] 250mm/sec FINE;
2955:L P[11013] 250mm/sec CNT100;
2956:L P[11014] 250mm/sec CNT100;
2957:L P[11015] 250mm/sec FINE;
2958:L P[11016] 250mm/sec CNT100;
2959:L P[11017] 250mm/sec CNT100;
2960:L P[11018] 250mm/sec FINE;
2961:L P[11019] 250mm/sec CNT100;
2962:L P[11020] 250mm/sec CNT100;
2963:L P[11021] 250mm/sec FINE;
2964:L P[11022] 250mm/sec CNT100;
2965:L P[11023] 250mm/sec CNT100;
2966:L P[11024] 250mm/sec FINE;
2967:L P[11025] 250mm/sec CNT100;
2968:L P[11026] 250mm/sec CNT100;
2969:L P[11027] 250mm/sec FINE;
2970:L P[11028] 250mm/sec CNT100;
2971:L P[11029] 250mm/sec CNT100;
2972:L P[11030] 250mm/sec FINE;
2973:L P[11031] 250mm/sec CNT100;
2974:L P[11032] 250mm/sec CNT100;
2975:L P[11033] 250mm/sec FINE;
2976:L P[11034] 250mm/sec CNT100;
2977:L P[11035] 250mm/sec CNT100;
2978:L P[11036] 250mm/sec FINE;
2979:L P[11037] 250mm/sec CNT100;
2980:L P[11038] 250mm/sec CNT100;
2981:L P[11039] 250mm/sec FINE;
2982:L P[11040] 250mm/sec CNT100;
2983:L P[11041] 250mm/sec CNT100;
2984:L P[11042] 250mm/sec FINE;
2985:L P[11043] 250mm/sec CNT100;
2986:L P[11044] 250mm/sec CNT100;
2987:L P[11045] 250mm/sec FINE;
2988:L P[11046] 250mm/sec CNT100;
2989:L P[11047] 250mm/sec CNT100;
2990:L P[11048] 250mm/sec FINE;
2991:L P[11049] 250mm/sec CNT100;
2992:L P[11050] 250mm/sec CNT100;
2993:L P[11051] 250mm/sec FINE;
2994:L P[11052] 250mm/sec CNT100;
2995:L P[11053] 250mm/sec CNT100;
2996:L P[11054] 250mm/sec FINE;
2997:L P[11055] 250mm/sec CNT100;
2998:L P[11056] 250mm/sec CNT100;
2999:L P[11057] 250mm/sec FINE;
3000:L P[11058] 250mm/sec CNT100;
3001:L P[11059] 250mm/sec CNT100;
3002:L P[11060] 250mm/sec FINE;
3003:L P[11061] 250mm/sec CNT100;
3004:L P[11062] 250mm/sec CNT100;
3005:L P[11063] 250mm/sec FINE;
3006:L P[11064] 250mm/sec CNT100;
3007:L P[11065] 250mm/sec CNT100;
3008:L P[11066] 250mm/sec FINE;
3009:L P[11067] 250mm/sec CNT100;
3010:L P[11068] 250mm/sec CNT100;
3011:L P[11069] 250mm/sec FINE;
3012:L P[11070] 250mm/sec CNT100;
3013:L P[11071] 250mm/sec CNT100;
3014:L P[11072] 250mm/sec FINE;
3015:L P[11073] 250mm/sec CNT100;
3016:L P[11074] 250mm/sec CNT100;
3017:L P[11075] 250mm/sec FINE;
3018:L P[11076] 250mm/sec CNT100;
3019:L P[11077] 250mm/sec CNT100;
3020:L P[11078] 250mm/sec FINE;
3021:L P[11079] 250mm/sec CNT100;
3022:L P[11080] 250mm/sec CNT100;
3023:L P[11081] 250mm/sec FINE;
3024:L P[11082] 250mm/sec CNT100;
3025:L P[11083] 250mm/sec CNT100;
3026:L P[11084] 250mm/sec FINE;
3027:L P[11085] 250mm/sec CNT100;
3028:L P[11086] 250mm/sec CNT100;
3029:L P[11087] 250mm/sec FINE;
3030:L P[11088] 250mm/sec CNT100;
3031:L P[11089] 250mm/sec CNT100;
3032:L P[11090] 250mm/sec FINE;
3033:L P[11091] 250mm/sec CNT100;
3034:L P[11092] 250mm/sec CNT100;
3035:L P[11093] 250mm/sec FINE;
3036:L P[11094] 250mm/sec CNT100;
3037:L P[11095] 250mm/sec CNT100;
3038:L P[11096] 250mm/sec FINE;
3039:L P[11097] 250mm/sec CNT100;
3040:L P[11098] 250mm/sec CNT100;
3041:L P[11099] 250mm/sec FINE;
3042:L P[11100] 250mm/sec CNT100;
3043:L P[11101] 250mm/sec CNT100;
3044:L P[11102] 250mm/sec FINE;
3045:L P[11103] 250mm/sec CNT100;
3046:L P[11104] 250mm/sec CNT100;
3047:L P[11105] 250mm/sec FINE;
3048:L P[11106] 250mm/sec CNT100;
3049:L P[11107] 250mm/sec CNT100;
3050:L P[11108] 250mm/sec FINE;
3051:L P[11109] 250mm/sec CNT100;
3052:L P[11110] 250mm/sec CNT100;
3053:L P[11111] 250mm/sec FINE;
3054:L P[11112] 250mm/sec CNT100;
3055:L P[11113] 250mm/sec CNT100;
3056:L P[11114] 250mm/sec FINE;
3057:L P[11115] 250mm/sec CNT100;
3058:L P[11116] 250mm/sec CNT100;
3059:L P[11117] 250mm/sec FINE;
3060:L P[11118] 250mm/sec CNT100;
3061:L P[11119] 250mm/sec CNT100;
3062:L P[11120] 250mm/sec FINE;
3063:L P[11121] 250mm/sec CNT100;
3064:L P[11122] 250mm/sec CNT100;
3065:L P[11123] 250mm/sec FINE;
3066:L P[11124] 250mm/sec CNT100;
3067:L P[11125] 250mm/sec CNT100;
3068:L P[11126] 250mm/sec FINE;
3069:L P[11127] 250mm/sec CNT100;
3070:L P[11128] 250mm/sec CNT100;
3071:L P[11129] 250mm/sec FINE;
3072:L P[11130] 250mm/sec CNT100;
